	ActCol				: DINT;
	ActVarConfig		: CSV_Config;
	ActVarValueString	: STRING;
	AdressOffset		: DINT;

	FPStart				: R_TRIG;
	FNStart				: F_TRIG;

	FBFileOpen			: FB_FileOpen;
	nOpenMode			: DWORD;
	hHandle				: UINT;

	CreateHeaderLineNow:BOOL;

	FBFileWrite			: FB_FileWrite;
	FBFileClose			: FB_FileClose;
	FileOpenWasBusy		: BOOL;
	FileWriteWasBusy	: BOOL;
	FileCloseWasBusy	: BOOL;
	FileOpenStart		: BOOL;
	FileWriteStart		: BOOL;
	FileCloseStart		: BOOL;

	TempString			: STRING[255];
END_VAR
FPStart(CLK:= nInExport );
FNStart(CLK:= nInExport );

IF 	FPStart.Q THEN
	WorkingStep:=1;
	FileOpenWasBusy:=FALSE;
	FileWriteWasBusy:=FALSE;
	FileCloseWasBusy:=FALSE;
	FileOpenStart:=FALSE;
	FileWriteStart:=FALSE;
	FileCloseStart:=FALSE;
	WorkingStepWriteLine:=1;
	TempString:='';
END_IF;

IF 	FNStart.Q AND WorkingStep<>50 THEN
	WorkingStep:=0;
END_IF


CASE WorkingStep OF

	1:	(* Check File Exist *)
		FindFile_.bExecute:=TRUE;
		IF 	FindFile_.bBusy THEN
			WorkingStep:=2;
		END_IF
	2:
		FindFile_.bExecute:=TRUE;
		IF 	NOT FindFile_.bBusy THEN
			WorkingStep:=3;
		END_IF
	3:
		IF  	filesList_.sFileName='' THEN
			(* Create Header *)
			WorkingStep:=20;
			CreateHeaderLineNow:=CreateHeaderLine;
		ELSIF
			filesList_.sFileName<>'' THEN
			(* File Exists *)
			WorkingStep:=20;
			CreateHeaderLineNow:=FALSE;
		END_IF

	20: (* Open File *)
		IF 	OverwriteExistingFile THEN
			nOpenMode:=FOPEN_MODEWRITE OR FOPEN_MODETEXT ;
		ELSE
			nOpenMode:=FOPEN_MODEAPPEND OR FOPEN_MODETEXT ;
		END_IF
		FBFileOpen(
			sNetId			:= localAMSNetID,
			sPathName	:= strInFileName,
			nMode			:= nOpenMode,
			ePath			:= PATH_GENERIC,
			bExecute		:= FileOpenStart,
			tTimeout		:= t#1s);
			hHandle:=FBFileOpen.hFile;
		FileOpenStart:= TRUE;
		IF 	FBFileOpen.bBusy THEN
			FileOpenWasBusy:=TRUE;
		END_IF
		IF 	NOT FBFileOpen.bBusy AND FileOpenWasBusy THEN
			WorkingStep:=21;
			FileOpenStart:= FALSE;
		END_IF

	21:	(* Write Header if required *)
		IF 	CreateHeaderLineNow THEN
			IF 	WorkingStepWriteLine=0 THEN
				WorkingStepWriteLine:=0;
				TempString:='';
			END_IF

			CASE WorkingStepWriteLine OF
				0: (*Create new CSV config*)
						WorkingStepWriteLine:=1;
				1: (* Open File *)
					FOR ActCol := 1 TO iInNumberOfColumns DO
						(*CSV-Configuration zuweisen*)
						ActVarConfig:=CSVConfig[ActCol];
						TempString:=CONCAT(TempString,ActVarConfig.ColName);
						IF 	ActCol<iInNumberOfColumns THEN
							TempString:=CONCAT(TempString,';');
						ELSE
							TempString:=CONCAT(TempString, '$N');
						END_IF
					END_FOR;
					WorkingStepWriteLine:=2;
				2:(* Write Line *)
				FBFileWrite(
					sNetId				:=localAMSNetID ,
					hFile				:=hHandle ,
					pWriteBuff			:=ADR(TempString) ,
					cbWriteLen			:=LEN(TempString) ,
					bExecute			:=FileWriteStart ,
					tTimeout				:=t#1s );
					FileWriteStart			:= TRUE;
	
				IF 	FBFileWrite.bBusy  THEN
					FileWriteWasBusy:=TRUE;
				END_IF
				IF 	(NOT FBFileWrite.bBusy) AND FileWriteWasBusy THEN
					FileWriteStart:= FALSE;
					FileWriteWasBusy:=FALSE;

					WorkingStepWriteLine:=0;
					WorkingStep:=30;
				END_IF
			END_CASE
		ELSE
			WorkingStep:=30;
		END_IF

	30:	(* Write Data *)
		IF 	WorkingStepWriteLine=0 THEN
			WorkingStepWriteLine:=0;
			TempString:='';
		END_IF

		CASE WorkingStepWriteLine OF
			0: (*Create new CSV config*)
					WorkingStepWriteLine:=1;
			1: (* Open File *)
				FOR ActCol := 1 TO iInNumberOfColumns DO
					(*CSV-Configuration zuweisen*)
					ActVarConfig:=CSVConfig[ActCol];
					AdressOffset:=0;
					ActVarValueString:=TYPEDEF_TO_STRING(ActVarConfig,AdressOffset);
					TempString:=CONCAT(TempString,ActVarValueString);
					IF 	ActCol<iInNumberOfColumns THEN
						TempString:=CONCAT(TempString,';');
					ELSE
						TempString:=CONCAT(TempString, '$N');
					END_IF
				END_FOR
				WorkingStepWriteLine:=2;
			2:(* Write Line *)
			FBFileWrite(
				sNetId				:=localAMSNetID ,
				hFile				:=hHandle ,
				pWriteBuff			:=ADR(TempString) ,
				cbWriteLen			:=LEN(TempString) ,
				bExecute			:=FileWriteStart ,
				tTimeout				:=t#1s );
				FileWriteStart			:= TRUE;

			IF 	FBFileWrite.bBusy  THEN
				FileWriteWasBusy:=TRUE;
			END_IF
			IF 	(NOT FBFileWrite.bBusy) AND FileWriteWasBusy THEN
				FileWriteStart:= FALSE;
				FileWriteWasBusy:=FALSE;

				WorkingStepWriteLine:=0;
				WorkingStep:=40;

			END_IF
		END_CASE

	40: (* Close File *)
		FBFileClose(
			sNetId:=localAMSNetID ,
			hFile:= hHandle,
			bExecute:=FileCloseStart ,
			tTimeout:= t#1s);
		FileCloseStart:=TRUE;
		IF 	FBFileClose.bBusy THEN
			FileCloseWasBusy:=TRUE;
		END_IF

		IF 	NOT FBFileClose.bBusy AND FileCloseWasBusy THEN
			WorkingStep:=50;
		END_IF
	50:(* Done *)
		Done:=TRUE;
		IF 	FNStart.Q THEN
			WorkingStep:=0;
			done:=FALSE;
		END_IF

END_CASE

FindFile_(
	sNetId:= '',
	sPathName:= strInFileName,
	stFindFile=> filesList_
);

FindFile_.bExecute:=FALSE;
END_FUNCTION_BLOCK

(* POU zLibrary/CSV_ImportExport/TYPEDEF_TO_STRING, ST *)
FUNCTION TYPEDEF_TO_STRING : STRING
VAR_INPUT
	TypeData				:CSV_Config;
	inAdressOffset			:DINT;
END_VAR
VAR
	pBOOL					:POINTER TO 	BOOL;
	pBYTE					:POINTER TO 	BYTE;
	pWORD				:POINTER TO 	WORD;
	pDWORD				:POINTER TO 	DWORD;
	pSINT					:POINTER TO 	SINT;
	pUSINT					:POINTER TO USINT;
	pINT					:POINTER TO INT;
	pUINT					:POINTER TO UINT;
	pDINT					:POINTER TO DINT;
	pUDINT				:POINTER TO UDINT;
	pREAL					:POINTER TO REAL;
	pLREAL				:POINTER TO LREAL;
	pSTRING				:POINTER TO STRING(255);
	pTIME					:POINTER TO TIME;
	pTOD					:POINTER TO TOD;
	pDATE					:POINTER TO DATE;
	pDT					:POINTER TO DT;
END_VAR
VAR CONSTANT
	TempTypeData			:DataTypeDef;
END_VAR
IF 	TypeData.ColDataType = TempTypeData.iBOOL THEN
	pBOOL:=TypeData.ColSourceAdr + inAdressOffset;
	TYPEDEF_TO_STRING:=BOOL_TO_STRING(pBOOL^);
ELSIF
	TypeData.ColDataType = TempTypeData.iBYTE THEN
	pBYTE:=TypeData.ColSourceAdr + inAdressOffset;
	TYPEDEF_TO_STRING:=BYTE_TO_STRING(pBYTE^);
ELSIF
	TypeData.ColDataType = TempTypeData.iWORD THEN
	pWORD:=TypeData.ColSourceAdr + inAdressOffset;
	TYPEDEF_TO_STRING:=WORD_TO_STRING(pWORD^);
ELSIF
	TypeData.ColDataType = TempTypeData.iDWORD THEN
	pDWORD:=TypeData.ColSourceAdr + inAdressOffset;
	TYPEDEF_TO_STRING:=DWORD_TO_STRING(pDWORD^);
ELSIF
	TypeData.ColDataType = TempTypeData.iSINT THEN
	pSINT:=TypeData.ColSourceAdr + inAdressOffset;
	TYPEDEF_TO_STRING:=SINT_TO_STRING(pSINT^);
ELSIF
	TypeData.ColDataType = TempTypeData.iUSINT THEN
	pUSINT:=TypeData.ColSourceAdr + inAdressOffset;
	TYPEDEF_TO_STRING:=USINT_TO_STRING(pUSINT^);
ELSIF
	TypeData.ColDataType = TempTypeData.iINT THEN
	pINT:=TypeData.ColSourceAdr + inAdressOffset;
	TYPEDEF_TO_STRING:=INT_TO_STRING(pINT^);
ELSIF
	TypeData.ColDataType = TempTypeData.iUINT THEN
	pUINT:=TypeData.ColSourceAdr + inAdressOffset;
	TYPEDEF_TO_STRING:=UINT_TO_STRING(pUINT^);
ELSIF
	TypeData.ColDataType = TempTypeData.iDINT THEN
	pDINT:=TypeData.ColSourceAdr + inAdressOffset;
	TYPEDEF_TO_STRING:=DINT_TO_STRING(pDINT^);
ELSIF
	TypeData.ColDataType = TempTypeData.iUDINT THEN
	pUDINT:=TypeData.ColSourceAdr + inAdressOffset;
	TYPEDEF_TO_STRING:=UDINT_TO_STRING(pUDINT^);
ELSIF
	TypeData.ColDataType = TempTypeData.iREAL THEN
	pREAL:=TypeData.ColSourceAdr + inAdressOffset;
	TYPEDEF_TO_STRING:=REAL_TO_STRING(pREAL^);
ELSIF
	TypeData.ColDataType = TempTypeData.iLREAL THEN
	pLREAL:=TypeData.ColSourceAdr + inAdressOffset;
	TYPEDEF_TO_STRING:=LREAL_TO_STRING(pLREAL^);
ELSIF
	TypeData.ColDataType = TempTypeData.iSTRING THEN
	pSTRING:=TypeData.ColSourceAdr + inAdressOffset;
	IF 	pSTRING^='' THEN
		TYPEDEF_TO_STRING:='empty';
	ELSE
		TYPEDEF_TO_STRING:=pSTRING^;
	END_IF
ELSIF
	TypeData.ColDataType = TempTypeData.iTIME THEN
	pTIME:=TypeData.ColSourceAdr + inAdressOffset;
	TYPEDEF_TO_STRING:=TIME_TO_STRING(pTIME^);
ELSIF
	TypeData.ColDataType = TempTypeData.iTOD THEN
	pTOD:=TypeData.ColSourceAdr + inAdressOffset;
	TYPEDEF_TO_STRING:=TOD_TO_STRING(pTOD^);
ELSIF
	TypeData.ColDataType = TempTypeData.iDATE THEN
	pDATE:=TypeData.ColSourceAdr + inAdressOffset;
	TYPEDEF_TO_STRING:=DATE_TO_STRING(pDATE^);
ELSIF
	TypeData.ColDataType = TempTypeData.iDT THEN
	pDT:=TypeData.ColSourceAdr + inAdressOffset;
	TYPEDEF_TO_STRING:=DT_TO_SPECIALSTRING(pDT^);
ELSE
	TYPEDEF_TO_STRING:='error';
END_IF
END_FUNCTION

(* POU zLibrary/CSV_ImportExport/DT_TO_SPECIALSTRING, ST *)
FUNCTION DT_TO_SPECIALSTRING : STRING
VAR_INPUT
	inDT			:DT;
END_VAR
VAR
	TempString		:STRING;
	SysTime		:TIMESTRUCT;

	wYear			:WORD;
	wMonth			:WORD;
	wDay			:WORD;
	wHour			:WORD;
	wMin			:WORD;
	wSec			:WORD;
END_VAR
SysTime:=DT_TO_SYSTEMTIME(inDT);
wYear:=SysTime.wYear;
wMonth:=SysTime.wMonth;
wDay:=SysTime.wDay;
wHour:=SysTime.wHour;
wMin:=SysTime.wMinute;
wSec:=SysTime.wSecond;
TempString:='';

IF 	wDay<10 THEN
	TempString:=CONCAT(TempString ,WORD_TO_STRING(0));
END_IF
TempString:=CONCAT(TempString ,WORD_TO_STRING(wDay));
TempString:=CONCAT(TempString , '.');
IF 	wMonth<10 THEN
	TempString:=CONCAT(TempString ,WORD_TO_STRING(0));
END_IF
TempString:=CONCAT(TempString ,WORD_TO_STRING(wMonth));
TempString:=CONCAT(TempString , '.');
TempString:=CONCAT(TempString ,WORD_TO_STRING(wYear));
TempString:=CONCAT(TempString , ' ');
IF 	wHour<10 THEN
	TempString:=CONCAT(TempString ,WORD_TO_STRING(0));
END_IF
TempString:=CONCAT(TempString ,WORD_TO_STRING(wHour));
TempString:=CONCAT(TempString , ':');
IF 	wMin<10 THEN
	TempString:=CONCAT(TempString ,WORD_TO_STRING(0));
END_IF
TempString:=CONCAT(TempString ,WORD_TO_STRING(wMin));
TempString:=CONCAT(TempString , ':');
IF	wSec<10 THEN
	TempString:=CONCAT(TempString ,WORD_TO_STRING(0));
END_IF
TempString:=CONCAT(TempString ,WORD_TO_STRING(wSec));
DT_TO_SPECIALSTRING:=TempString;
END_FUNCTION

(* POU System/Error_and_Message/MessageHandler, ST *)
PROGRAM MessageHandler
VAR_INPUT
	Prio					: DINT; 					(*1=highest, .. , 4=lowest*)
	Btn1Addr 			: POINTER TO BOOL;	(*Address of Button1 , if Zero then Button is unvisible*)
	Btn2Addr 			: POINTER TO BOOL;	(*Address of Button2 , if Zero then Button is unvisible*)
	Msg				: sMessageText;
	MessageLine		: ARRAY [1..10] OF sMessageLine;
	MsgButton1Text		: STRING(20);
	MsgButton2Text		: STRING(20);

	FB_ReadXmlLineMsg	:FB_ReadXmlLine;
END_VAR
VAR_IN_OUT
	sVisu				: sMessageVisu;
END_VAR
VAR_OUTPUT
	MessageActive		: BOOL;
END_VAR
VAR
	EmptyMsg			: sMessageText;
	TempMsg			: sMessageText;
	TempPrio			: DINT;
	MessageGoneFlag	: F_TRIG;
	MessageShowFlag	: R_TRIG;
	Idx, i					: DINT;
	BackupVisu			: STRING;
	ShowVisuMessage	: BOOL;
	VisuMessageActivT	: TON;

	Button1				: VisuButton;
	Button2				: VisuButton;
	btnHide				: VisuButton;
	btnShow			: VisuButton;
	ShowText			: STRING(255);
	LaufschriftShowText	: FB_Laufschrift_STR255;

(* Vars for Disabling Multiselection *)
	Index			: DINT;
	Index_Clear			: DINT;
	FP_MsgLineBool	: ARRAY[1..20] OF R_TRIG;
	LastPressedLine		: DINT;

	Error				: ErrorStruct;
	ErrorPuls			: BOOL:=FALSE;

END_VAR
(*Das ist noch Baustelle!
Es gibt 2 Möglichkeiten:
a) Prio bei Messages mit Button gibt es nicht.
   Wenn eine Meldung mit Button angezeigt wird, dann solange bis diese quittiert ist.
   Dann erst kommt die nächste dran.

b) Jede Meldung mit Button erhält eine eindeutige PLCID.
   Die Visu schreibt für die angezeigte Meldung die ID zurück in VisuID.
   Wenn das Button-Signal in der PLC ankommt werden die IDs verglichen,
   und nur bei VisuID=PLCID wird der Button an die Aufrufstelle weitergereicht.
*)

Lng();

IF 	(NOT TempMsg.ShowMessage OR
	 Msg.Name=TempMsg.Name AND Msg.Text=TempMsg.Text) THEN
	IF 	Msg.Name=TempMsg.Name	AND
		Msg.Text=TempMsg.Text THEN
		IF 	Btn1Addr<>0 THEN
			IF 	MsgButton1Text='' THEN
				MsgButton1Text:='OK';
			END_IF
			Button1.Enable:=TRUE;
			Button1.Visible:=TRUE;
			Button1.TextOn:=MsgButton1Text;
			IF 	sVisu.Button1.Pressed THEN
				Btn1Addr^:=TRUE;
				MessageLine:=sVisu.MessageLine;
				TempMsg.ShowMessage:=FALSE;
			END_IF
		ELSE
			Button1.Visible:=FALSE;
		END_IF

		IF 	Btn2Addr<>0 THEN
			IF 	MsgButton2Text='' THEN
				MsgButton2Text:='Cancel';
			END_IF
			Button2.Enable:=TRUE;
			Button2.Visible:=TRUE;
			Button2.TextOn:=MsgButton2Text;
			IF 	sVisu.Button2.Pressed THEN
				Btn2Addr^:=TRUE;
				TempMsg.ShowMessage:=FALSE;
			END_IF
		ELSE
			Button2.Visible:=FALSE;
		END_IF
	ELSE
		TempMsg:=Msg;
		sVisu.MessageLine:=MessageLine;
	END_IF
	TempMsg.ShowMessage:=TRUE;
	TempPrio:=Prio;

	IF 	NOT ErrorPuls OR
		Error.DateTime = ErrorHandler.EmptyError.DateTime THEN
		Error.DateTime	:= gVarDTSystemtime;
		ErrorPuls 		:= TRUE;
	END_IF
	Error.Text	:= CONCAT('MessageHandler: ',Msg.Text);
	Error.No		:= 1;
	Error.Typ	:= 1;			(* 0=red 1:=orange 2:=blue *)

	IF 	Error.Text<>'' AND
		ST_Lng.b_EndChangeLng THEN
		ErrorHandler.AddError(	ErrorToAdd:=Error,
								sVisu:=Visu.ErrorHandler);
	END_IF
END_IF


(*Clear Input-Var*)
Prio:=0;
Btn1Addr:=0;
Btn2Addr:=0;
Msg:=EmptyMsg;
MsgButton1Text:='';
MsgButton2Text:='';
END_PROGRAM
ACTION ClearAll:
IF NOT sVisu.ShowMessage THEN
	TempPrio:=0;
	TempMsg.Name:='';
	TempMsg.Text:='';
	TempMsg.ID:='';
	TempMsg.ShowMessage:=FALSE;
	TempMsg.Color:=0;
	TempMsg.Station:=0;
	TempMsg.Button1.Visible:=FALSE;
	TempMsg.Button2.Visible:=FALSE;
ELSE
	TempMsg.ShowMessage:=FALSE;
END_IF

(* Copy from visu *)
MessageLine:=sVisu.MessageLine;
END_ACTION
ACTION ClearMessageLines:
FOR idx:=1 TO 10 DO
	MessageHandler.MessageLine[idx].Visible:=FALSE;
	MessageHandler.MessageLine[idx].Editable:=FALSE;
	MessageHandler.MessageLine[idx].Text:='';
	MessageHandler.MessageLine[idx].MsgInt:=0;
	MessageHandler.MessageLine[idx].MsgBool:=FALSE;
	MessageHandler.MessageLine[idx].MsgReal:=0.0;
	MessageHandler.MessageLine[idx].MsgString:='';
	MessageHandler.MessageLine[idx].MsgTypeEnum:=MsgDataTypeNone;
END_FOR
END_ACTION
ACTION DisableMultiSelect:
LastPressedLine:=0;

FOR Index:=1 TO 10 DO
	FP_MsgLineBool[Index](CLK:=sVisu.MessageLine[Index].MsgBool);
	IF FP_MsgLineBool[Index].Q THEN
		LastPressedLine:=Index;
		EXIT;
	END_IF
END_FOR

IF LastPressedLine>0 THEN

	FOR Index_Clear:=1 TO 10 DO
		MessageLine[Index_Clear].MsgBool:=(LastPressedLine=Index_Clear);
	END_FOR

END_IF
END_ACTION
ACTION Lng:
IF	TempMsg.ID <> '' THEN

	FB_ReadXmlLineMsg(
		Prefix:= 'MSG',
		ID:= TempMsg.ID,
		File:= 'MSG.xml',
		Text=>);

	IF 	FB_ReadXmlLineMsg.Text <> ''  THEN
		TempMsg.Text:=CONCAT(TempMsg.ID,':$N$R');
		TempMsg.Text:=CONCAT(TempMsg.Text,FB_ReadXmlLineMsg.Text);
		Msg.Text:=TempMsg.Text;

		ShowText:=CONCAT(TempMsg.ID,': ');
		ShowText:=CONCAT(ShowText,FB_ReadXmlLineMsg.Text);
		FOR i:=1 TO 10 DO
			IF	FIND(ShowText, '$N') > 0 THEN
				ShowText:=DELETE (ShowText,1,FIND(ShowText, '$N'));
			END_IF
			IF	FIND(ShowText, '$R') > 0 THEN
				ShowText:=DELETE (ShowText,1,FIND(ShowText, '$R'));
			END_IF
		END_FOR
		IF LEN(ShowText) > 60 THEN
			ShowText:=CONCAT(ShowText,' ->   ');
		END_IF
		LaufschriftShowText(
				N:= 60,
				StepWidth:=1,
				PT:= t#100ms ,
				Text:= ShowText,
				Display=>BtnShow.TextOn
				);
	ELSE
		TempMsg.Text:=CONCAT(TempMsg.ID,':..... ');
	END_IF
ELSE
	ShowText:=TempMsg.Text;
	FOR i:=1 TO 10 DO
		IF	FIND(ShowText, '$N') > 0 THEN
			ShowText:=DELETE (ShowText,1,FIND(ShowText, '$N'));
		END_IF
		IF	FIND(ShowText, '$R') > 0 THEN
			ShowText:=DELETE (ShowText,1,FIND(ShowText, '$R'));
		END_IF
	END_FOR
	IF LEN(ShowText) > 60 THEN
		ShowText:=CONCAT(ShowText,' ->   ');
	END_IF
	LaufschriftShowText(
			N:= 60,
			StepWidth:=1,
			PT:= t#100ms ,
			Text:= ShowText,
			Display=>BtnShow.TextOn
			);
END_IF
END_ACTION
ACTION VisuUpdate:
sVisu.Name:=TempMsg.Name;
sVisu.Text:=TempMsg.Text;
sVisu.ID:=TempMsg.ID;
sVisu.ShowMessage:=TempMsg.ShowMessage;
sVisu.Color:=TempMsg.Color;
sVisu.Station:=TempMsg.Station;

sVisu.Button1:=TempMsg.Button1;
sVisu.Button2:=TempMsg.Button2;


(* Write to visu *)

sVisu.MessageLine:=MessageLine;
FOR idx:=1 TO 10 DO
	CASE sVisu.MessageLine[idx].MsgTypeEnum OF
		MsgDataTypeBool: sVisu.MessageLine[idx].MsgType:='BOOL';
		MsgDataTypeDint: sVisu.MessageLine[idx].MsgType:='DINT';
		MsgDataTypeReal: sVisu.MessageLine[idx].MsgType:='REAL';
		MsgDataTypeString: sVisu.MessageLine[idx].MsgType:='STRING';
	ELSE
		sVisu.MessageLine[idx].MsgType:='';
	END_CASE
END_FOR

MessageGoneFlag(CLK:=sVisu.ShowMessage);
MessageShowFlag(CLK:=sVisu.ShowMessage AND NOT sVisu.BtnShow.Pressed);

(*Meldefenster öffnen, wenn Meldung neu aktiv wird (als Impuls)*)
IF MessageShowFlag.Q AND CurrentVisu<>'ZLIB_VISUMESSAGEHANDLER' THEN
	ShowVisuMessage:=TRUE;
	BackupVisu:=CurrentVisu;
END_IF
VisuMessageActivT(IN:=CurrentVisu='ZLIB_VISUMESSAGEHANDLER' ,PT:=T#1s);
IF 	CurrentVisu='ZLIB_VISUMESSAGEHANDLER'AND
	ShowVisuMessage THEN
	ShowVisuMessage:=FALSE;
END_IF
IF 	ShowVisuMessage THEN
	CurrentVisu:='ZLIB_VISUMESSAGEHANDLER';
END_IF

(*Button "Meldung einblenden" anzeigen, wenn Meldung aktiv aber Meldefenster nicht offen*)
IF 	sVisu.ShowMessage AND
	CurrentVisu<>'ZLIB_VISUMESSAGEHANDLER' AND
	NOT ShowVisuMessage THEN
	BtnShow.Visible:=TRUE;
	BtnShow.Enable:=TRUE;
	BtnShow.ButtBackColor:=Visu.Message.Color;
ELSE
	BtnShow.Visible:=FALSE;
END_IF

(*Button "Minimieren" einblenden, wenn Meldefenster offen*)
IF 	CurrentVisu='ZLIB_VISUMESSAGEHANDLER' THEN
	BtnHide.Visible:=TRUE;
	BtnHide.Enable:=TRUE;
	BtnHide.TextOn:='Meldung minimieren';
	BtnHide.ButtBackColor:=Color.control;
ELSE
	BtnHide.Visible:=FALSE;
END_IF

(*Meldefenster komplett schliessen, wenn keine Meldung mehr ansteht*)
IF 	MessageGoneFlag.Q OR
	BtnHide.Pressed THEN
	IF 	BackupVisu<>'' OR
		BackupVisu='ZLIBVISUMESSAGEHANDLER'THEN
		CurrentVisu:=BackupVisu;
	ELSE
		CurrentVisu:='MAIN';
	END_IF
END_IF;

MessageActive := sVisu.ShowMessage OR sVisu.BtnShow.Visible;


(*VisuButton Handler Call*)
Button1(	Button:= TempMsg.Button1);
Button2(	Button:= TempMsg.Button2);
btnHide(	Button:= sVisu.btnHide);
btnShow(	Button:= sVisu.btnShow);
END_ACTION

(* POU zLibrary/ept/Sprache/FB_ReadXmlLine, ST *)
FUNCTION_BLOCK FB_ReadXmlLine
VAR_INPUT
	Prefix					: STRING;
	ID						: STRING;
	File						: STRING;
END_VAR
VAR_OUTPUT
	Text					: STRING(255);
END_VAR

VAR
	bError							: BOOL;
	nErrId							: UDINT;

	fb_state_entry					: ST_StateEntry;

	CURRENTLANGUAGECopy			: STRING(5);
	IdCopy							: STRING;
END_VAR
(*======================================================
   ST: FB_ReadXmlLine
 ------------------------------------------------------
   Auth: 	Werner Frield    						 
   Date: 	23.12.2020    						     
   Rev.: 		1.0	
   Desc	
	-	Mit diesem FB kann Srachabängig ein Text aus einer xml Datei ausgelesen werden		
	-	Das Programm ST_ReadXmlLine wird zum auslesen benutzt.
	-	Die XML Datei muss im PLC Verzeichnis unter TRANS abgelegt werden und 
		mit der Excel Datei (_Texte.xlsm) erstellt werden.
	-	abhängig von der CURRENTLANGUAGE werden Srachabängig die Texte ausgelesen

Beispiel:
FB_ReadXmlLineConf(
	Prefix:= 'CONFIG',			(*erste Spalte der Excel Datei*)
	ID:= 'ST03_473_B70_0',		(*zweite Spalte der Excel Datei*)
	File:= 'CONFIG.xml',		(* xml Datei Name*)
	Text=> );					(* hier kommt der passende Text zurück. abhängig von der angewählten Sprache (DE, EN,CZ*)

 ========================================================*)
fb_state_entry(i16_pos:= 1);
CASE fb_state_entry.i16_step OF
(*=======================================================*)
INIT_OBJ:

	(*-----------------------Weiterschaltbedingungen----------------------------*)
	fb_state_entry.i16_next_step:=INIT;

(*=======================================================*)
INIT:
	IF	TD.ArtNo <> '' AND CURRENTLANGUAGE <> '' THEN
		fb_state_entry.i16_next_step:=BEREIT;
	END_IF

(*=======================================================*)
BEREIT:	fb_state_entry.s_debugtext:='warte auf Start';

	IF	fb_state_entry.E THEN
		bError:=FALSE;
		IdCopy:= ID;
	END_IF
	IF	Prefix <> '' AND ID <> '' AND
		ST_ReadXmlLine.b_ready THEN

		IF	CURRENTLANGUAGECopy <> CURRENTLANGUAGE OR
			IdCopy <> ID THEN
			IF	Prefix <> 'MSG' THEN
				fb_state_entry.i16_next_step:=110;		(*ST_ReadXmlLine*)
			ELSE
				fb_state_entry.i16_next_step:=210;		(*ST_ReadXmlLineMsg*)
			END_IF
		END_IF
	END_IF

	IF	fb_state_entry.X THEN
		CURRENTLANGUAGECopy := CURRENTLANGUAGE;
		Text:='';
	END_IF

(*=======================================================*)
110:  fb_state_entry.s_debugtext:='*Warten bis Lesen erlaubt ist';

	IF	TestAndSet(ST_ReadXmlLine.LockFlag) THEN
		fb_state_entry.i16_next_step := 120;
	END_IF

	IF	fb_state_entry.X THEN
		ST_ReadXmlLine.b_start:=TRUE;
		ST_ReadXmlLine.s_Prefix:= Prefix;
		ST_ReadXmlLine.s_ID:= ID;
		ST_ReadXmlLine.s_File:= File;
		ST_ReadXmlLine.s_Text;
	END_IF

(*=======================================================*)
120:  fb_state_entry.s_debugtext:='*Warten auf busy';

	IF 	ST_ReadXmlLine.b_busy THEN
		fb_state_entry.i16_next_step := 130;
	ELSIF
		fb_state_entry.fb_ton_Step.ET > t#3000ms THEN
		nErrId := ST_ReadXmlLine.nErrId;
		fb_state_entry.s_debugtext:='timeout';
		fb_state_entry.i16_next_step := FEHLER;
	END_IF

(*=======================================================*)
130:  fb_state_entry.s_debugtext:='*Warten auf fertig';

	IF 	ST_ReadXmlLine.b_done THEN
		text:=ST_ReadXmlLine.s_Text;

		fb_state_entry.i16_next_step := BEREIT;
	ELSIF
		fb_state_entry.fb_ton_Step.ET > t#3000ms THEN
		nErrId := ST_ReadXmlLine.nErrId;
		fb_state_entry.s_debugtext:='timeout';
		fb_state_entry.i16_next_step := FEHLER;
	END_IF

(*=======================================================*)
(*=======================================================*)
210:  fb_state_entry.s_debugtext:='*Warten bis Lesen erlaubt ist';

	IF	TestAndSet(ST_ReadXmlLineMsg.LockFlag) THEN
		fb_state_entry.i16_next_step := 220;
	END_IF

	IF	fb_state_entry.X THEN
		ST_ReadXmlLineMsg.b_start:=TRUE;
		ST_ReadXmlLineMsg.s_Prefix:= Prefix;
		ST_ReadXmlLineMsg.s_ID:= ID;
		ST_ReadXmlLineMsg.s_File:= File;
		ST_ReadXmlLineMsg.s_Text;
	END_IF

(*=======================================================*)
220:  fb_state_entry.s_debugtext:='*Warten auf busy';

	IF 	ST_ReadXmlLineMsg.b_busy THEN
		fb_state_entry.i16_next_step := 230;
	ELSIF
		fb_state_entry.fb_ton_Step.ET > t#3000ms THEN
		nErrId := ST_ReadXmlLineMsg.nErrId;
		fb_state_entry.s_debugtext:='timeout';
		fb_state_entry.i16_next_step := FEHLER;
	END_IF

(*=======================================================*)
230:  fb_state_entry.s_debugtext:='*Warten auf fertig';

	IF 	ST_ReadXmlLineMsg.b_done THEN
		text:=ST_ReadXmlLineMsg.s_Text;
		fb_state_entry.i16_next_step := BEREIT;
	ELSIF
		fb_state_entry.fb_ton_Step.ET > t#3000ms THEN
		nErrId := ST_ReadXmlLineMsg.nErrId;
		fb_state_entry.s_debugtext:='timeout';
		fb_state_entry.i16_next_step := FEHLER;
	END_IF

(*=======================================================*)
FEHLER:
	IF 	fb_state_entry.E THEN
		bError:=TRUE;
		Text:=ST_ReadXmlLine.s_Text;
	END_IF

	fb_state_entry.s_debugtext:='nErrorID: ';
	fb_state_entry.s_debugtext:=CONCAT(fb_state_entry.s_debugtext, UDINT_TO_STRING(nErrId));
	fb_state_entry.i16_next_step:=BEREIT;

END_CASE
fb_state_entry(i16_pos:= 2);
END_FUNCTION_BLOCK

(* POU zLibrary/ept/Funktionsbausteine/ST_StateEntry, ST *)
FUNCTION_BLOCK ST_StateEntry
VAR
	arr_last_step_history	: ARRAY[0..31] OF STRING(110);
	last_pos 			: INT := 0;
	interner_step		: INT := 0;
	s_stepTime 			: STRING;
END_VAR
VAR_OUTPUT
	i16_last_step 			: enum_step_nr := INIT_OBJ;	(* Der Schritt vor diesem Schritt *)
	i16_step 				: enum_step_nr := INIT_OBJ;	(* Diese variable soll vom "case step of" verwendet werden *)
	E					: BOOL;					(* Aktiv bei betreten des Steps *)
	X					: BOOL;					(* Aktiv beim verlassen des Steps *)
	b_error 				: BOOL := FALSE;			(* Ablauf Pos 1,2,1,2,1,2,... nicht richtig *)
	fb_ton_Step			: TON;
END_VAR
VAR_INPUT
	i16_next_step 		: enum_step_nr := INIT_OBJ;	(* Nächster schritt *)
	i16_pos 				: INT;					(* Pos = 1: Aufruf vor dem Case step of ---  Pos = 2: Aufruf nach dem Case step of*)
	s_debugtext			: STRING(100);
END_VAR
VAR_TEMP
	i					: INT := 0;
END_VAR
VAR CONSTANT
	t_MaxStepTime		: TIME := T#60S;
END_VAR
(*stepTime ermitteln*)
fb_ton_Step(IN:= , PT:=fb_ton_Step.ET + t#10s , Q=>  , ET=> );
IF	i16_step = i16_next_step THEN
	fb_ton_Step.IN:=TRUE;
END_IF

IF	NOT b_error THEN
	CASE interner_step OF
		0:
			(* Mitten im Schritt drin *)
			X := FALSE;
			E := FALSE;


			(* Schritt wird verlassen *)
			IF i16_step <> i16_next_step AND i16_pos = 1 THEN
				subrDebugtext();
				interner_step := 10;
				X := TRUE;
				E := FALSE;
				fb_ton_Step.IN:=FALSE;
			END_IF

		10:
			(* Eintritt in neuen Schritt *)
			IF i16_pos = 1 THEN
				X := FALSE;
				E := TRUE;

				(* Schalte Schritt weiter *)
				i16_last_step := i16_step;
				i16_step := i16_next_step;
				(* Baue Statehistory *)

				IF  E THEN
					FOR i:= 31 TO 1 BY -1 DO
						arr_last_step_history[i] := arr_last_step_history[i-1];
					END_FOR
					arr_last_step_history[0] := '';
					s_stepTime:='';
					s_debugtext:='';
				END_IF

				interner_step := 0;

			END_IF
	END_CASE
END_IF

IF 	(fb_ton_Step.ET >= T#200ms AND arr_last_step_history[0] = '') OR	(* Am Anfang Debugtext schreiben, damit etwas drin steht *)
	(fb_ton_Step.Q AND s_stepTime <> '>1m') THEN	(* Debugtext schreiben, wenn t_MaxStepTime erreicht wird *)
	subrDebugtext();
END_IF

(* Prüfe Baustein *)
IF 	i16_pos = last_pos THEN
	b_error := TRUE;
END_IF

last_pos := i16_pos;
END_FUNCTION_BLOCK
ACTION subrDebugtext:
s_stepTime:=ET_TO_STRING(fb_ton_Step.ET);
IF 	fb_ton_Step.ET >= t_MaxStepTime THEN
	s_stepTime:=CONCAT('>',s_StepTime);
END_IF

(* history zusammenbauen aus StepNr, StepTime und debugtext*)
CASE i16_step OF
	INIT_OBJ :			arr_last_step_history[0]:='INIT_OBJ';
	INIT :				arr_last_step_history[0]:='INIT';
	BEREIT :			arr_last_step_history[0]:='BEREIT';
	HALT :				arr_last_step_history[0]:='HALT';
	STOP :				arr_last_step_history[0]:='STOP';
	FEHLER :			arr_last_step_history[0]:='FEHLER';
	INAKTIV:			arr_last_step_history[0]:='INAKTIV ';
ELSE
	arr_last_step_history[0] := INT_TO_STRING(i16_step);
END_CASE

IF 	s_stepTime ='0ms' OR s_stepTime =''THEN
	s_stepTime:='3ms';		(*damit nicht 0 drin steht*)
END_IF
arr_last_step_history[0] := CONCAT(arr_last_step_history[0],':  ');
arr_last_step_history[0] := CONCAT(arr_last_step_history[0],s_stepTime);
arr_last_step_history[0] := CONCAT(arr_last_step_history[0],': ');
arr_last_step_history[0] := CONCAT(arr_last_step_history[0],s_debugtext);
END_ACTION

(* POU zLibrary/ept/Funktionen/ET_TO_STRING, ST *)
FUNCTION ET_TO_STRING :STRING
VAR_INPUT
	et		:TIME;
END_VAR

VAR

END_VAR
ET_TO_STRING:=TIME_TO_STRING(et);
ET_TO_STRING:=DELETE(ET_TO_STRING,2,1);
END_FUNCTION

(* POU zLibrary/ept/Sprache/ST_ReadXmlLine, ST *)
PROGRAM ST_ReadXmlLine (*Programm wird nur vom FB_ReadXmlLine benutzt*)
VAR_INPUT
	b_start					: BOOL;
	s_Prefix					: STRING;
	s_ID					: STRING;
	s_File					: STRING;
	s_XmlHelp				: T_MaxString;	(* in diese Variable schreibt der XML-Bautstein die ausgelesenen Daten *)
END_VAR
VAR_OUTPUT
	b_EndChangeLng		: BOOL;
	b_busy					: BOOL;
	b_ready					: BOOL;
	b_done					: BOOL;

	s_Text					: STRING(255);
END_VAR

VAR

	LockFlag						: BOOL := FALSE;	(* Ganz wichtig, wenn diese Variable TRUE ist, dann kann die Struktur "Visu.MeldungProduktion" nicht verändert werden *)
	b_Error							: BOOL;
	nErrId							: UDINT;
	s_filePath						: T_MaxString;
	s_Xpath							: T_MaxString;

	fb_state_entry					: ST_StateEntry;
	fb_xml_srv_read					: FB_XmlSrvReadByName;	(* XML Baustein zum Auslesen der CONFIG *)

	CURRENTLANGUAGECopy			: STRING(5);
END_VAR
VAR CONSTANT
	s_SymName					: STRING:='ST_ReadXmlLine.s_XmlHelp';
END_VAR
(*Programm wird nur vom FB_ReadXmlLine benutzt*)

(*===================================================================================================*)
fb_state_entry(i16_pos:= 1);

CASE fb_state_entry.i16_step OF
(*=======================================================*)
INIT_OBJ:

	fb_state_entry.i16_next_step:=INIT;

(*=======================================================*)
INIT:

	IF	TD.ArtNo <> '' THEN
		fb_state_entry.i16_next_step:=BEREIT;
	END_IF

(*=======================================================*)
BEREIT:	fb_state_entry.s_debugtext:='warte auf Start';

	IF	fb_state_entry.E THEN
		b_Error:=FALSE;
		b_ready:=TRUE;
		LockFree();
	END_IF

	IF	s_Prefix <> '' AND s_ID <> '' AND
		b_start THEN
		fb_state_entry.i16_next_step:=110;
(*		LockGet();	(* Ablauf ist immer derselbe, zuerst LockGet, dann Strukturen ändern, dann LockFree *)*)
	END_IF

	IF	fb_state_entry.fb_ton_Step.ET >t#10ms THEN
		b_EndChangeLng:=TRUE;
	END_IF

	IF	fb_state_entry.X THEN
		IF 	CURRENTLANGUAGECopy<>CURRENTLANGUAGE THEN
			CURRENTLANGUAGECopy:=CURRENTLANGUAGE;
			b_EndChangeLng:=FALSE;
		END_IF
		s_XmlHelp:='';
		s_Text:='';
		b_ready:=FALSE;
		b_done:=FALSE;
		b_busy:=TRUE;
	END_IF

(*=======================================================*)
110:	fb_state_entry.s_debugtext:='Zeile aus der XMl auslesen';

	IF	fb_state_entry.E THEN
		s_filePath := CONCAT(s_PLC_path,'TRANS\');
		s_filePath := CONCAT(s_filePath,s_File);

		s_Xpath:= '/dynamic-text/text-list/text[@prefix=$'';
		s_Xpath:=CONCAT(s_Xpath,s_Prefix);
		s_Xpath:=CONCAT(s_Xpath,'$' and @id=$'');
		s_Xpath:=CONCAT(s_Xpath,s_ID);
		s_Xpath:=CONCAT(s_Xpath,'$']/');
		s_Xpath:=CONCAT(s_Xpath, CURRENTLANGUAGE);
	END_IF

	(*-----------------------Weiterschaltbedingungen----------------------------*)
	fb_state_entry.i16_next_step := 120;

(*=======================================================*)
120:	fb_state_entry.s_debugtext:='Starte Daten lesen ';

	IF 	fb_state_entry.E THEN
		fb_xml_srv_read.sFilePath := s_filePath;
		fb_xml_srv_read.sXPath :=s_Xpath;
		fb_xml_srv_read.sSymName := s_SymName;
		fb_xml_srv_read.bExecute := TRUE;
	END_IF

	(*-----------------------Weiterschaltbedingungen----------------------------*)
	IF 	fb_xml_srv_read.bBusy THEN
		fb_xml_srv_read.bExecute := FALSE;
		fb_state_entry.i16_next_step := 130;
	END_IF

(*=======================================================*)
130:fb_state_entry.s_debugtext:='warte auf fertig';

	(*-----------------------Weiterschaltbedingungen----------------------------*)
	IF  	NOT fb_xml_srv_read.bBusy  THEN
		fb_state_entry.i16_next_step := 140;
	ELSIF
		fb_state_entry.fb_ton_Step.ET > t#3000ms THEN
		nErrId := fb_xml_srv_read.nErrId;
		fb_state_entry.s_debugtext:='timeout';
		fb_state_entry.i16_next_step := FEHLER;
	END_IF

(*=======================================================*)
140:fb_state_entry.s_debugtext:='prüfe auf Fehler';

	(*-----------------------Weiterschaltbedingungen----------------------------*)
	IF  	fb_xml_srv_read.bError OR
		s_XmlHelp = '' THEN
		nErrId := fb_xml_srv_read.nErrId;
		fb_state_entry.i16_next_step := FEHLER;
	ELSE
		s_Text:=s_XmlHelp;
		fb_state_entry.i16_next_step := BEREIT;
		b_done:=TRUE;
		b_busy:=FALSE;
	END_IF


(*=======================================================*)
FEHLER:
	IF 	fb_state_entry.E THEN
		b_Error:=TRUE;
		s_Text:='!!! ';
		s_Text:= CONCAT(s_Text,s_Prefix);
		s_Text:= CONCAT(s_Text,'-');
		s_Text:= CONCAT(s_Text,s_ID);
		s_Text:= CONCAT(s_Text,' not found !!!');
	END_IF

	fb_state_entry.s_debugtext:='nErrorID: ';
	fb_state_entry.s_debugtext:=CONCAT(fb_state_entry.s_debugtext, UDINT_TO_STRING(nErrId));
	fb_state_entry.s_debugtext:=CONCAT(fb_state_entry.s_debugtext, ' =>');
	fb_state_entry.s_debugtext:=CONCAT(fb_state_entry.s_debugtext, s_Text);

	(*-----------------------Weiterschaltbedingungen----------------------------*)
	fb_state_entry.i16_next_step:=BEREIT;

	IF 	fb_state_entry.E THEN
		b_done:=TRUE;
		b_busy:=FALSE;
	END_IF

END_CASE

fb_state_entry(i16_pos:= 2);

b_start:=FALSE;


(* XML *)
fb_xml_srv_read(
	sNetId:= '',
	ePath:= PATH_GENERIC,
	nMode:= XMLSRV_SKIPMISSING,
	sSymName:= ,
	sFilePath:= ,
	sXPath:= ,
	bExecute:= ,
	tTimeout:= t#10s,
	bBusy=> ,
	bError=> ,
	nErrId=> );
END_PROGRAM
ACTION LockFree:
LockFlag := FALSE;	(* wieder freigeben *)
END_ACTION
ACTION LockGet:
WHILE NOT TestAndSet(LockFlag) DO	(* Mit der Funktion TestAndSet kann ein Flag nicht unterbrechbar geprüft und gesetzt werden *)
	;	(* Wait until Lock is free *)
END_WHILE
(*LockFlag: Ist ein boolsches Flag, das geprüft wird
 - war es FALSE, dann war das Flag frei und wird gesetzt (blockiert von nun an), die Funktion liefert TRUE
 - war es TRUE, dann war das Flag bereits belegt (blockiert), die Funktion liefert FALSE*)
END_ACTION

(* POU zLibrary/ept/Sprache/ST_ReadXmlLineMsg, ST *)
PROGRAM ST_ReadXmlLineMsg
VAR_INPUT
	b_start					: BOOL;
	s_Prefix					: STRING;
	s_ID					: STRING;
	s_File					: STRING;
	s_XmlHelp				: T_MaxString;	(* in diese Variable schreibt der XML-Bautstein die ausgelesenen Daten *)
END_VAR
VAR_OUTPUT
	b_EndChangeLng		: BOOL;
	b_busy					: BOOL;
	b_ready					: BOOL;
	b_done					: BOOL;

	s_Text					: STRING(255);
END_VAR

VAR
	LockFlag						: BOOL := FALSE;	(* Ganz wichtig, wenn diese Variable TRUE ist, dann kann die Struktur "Visu.MeldungProduktion" nicht verändert werden *)
	b_Error							: BOOL;
	nErrId							: UDINT;
	s_filePath						: T_MaxString;
	s_Xpath							: T_MaxString;

	fb_state_entry					: ST_StateEntry;
	fb_xml_srv_read					: FB_XmlSrvReadByName;	(* XML Baustein zum Auslesen der CONFIG *)

	CURRENTLANGUAGECopy			: STRING(5);
END_VAR
VAR CONSTANT
	s_SymName					: STRING:='ST_ReadXmlLineMsg.s_XmlHelp';
END_VAR
(*===================================================================================================*)
fb_state_entry(i16_pos:= 1);

CASE fb_state_entry.i16_step OF
(*=======================================================*)
INIT_OBJ:

	fb_state_entry.i16_next_step:=INIT;

(*=======================================================*)
INIT:

	IF	TD.ArtNo <> '' THEN
		fb_state_entry.i16_next_step:=BEREIT;
	END_IF

(*=======================================================*)
BEREIT:	fb_state_entry.s_debugtext:='warte auf Start';

	IF	fb_state_entry.E THEN
		b_Error:=FALSE;
		b_ready:=TRUE;
		LockFree();
	END_IF

	IF	s_Prefix <> '' AND s_ID <> '' AND
		b_start THEN
		fb_state_entry.i16_next_step:=110;
(*		LockGet();	(* Ablauf ist immer derselbe, zuerst LockGet, dann Strukturen ändern, dann LockFree *)*)
	END_IF

	IF	fb_state_entry.fb_ton_Step.ET >t#10ms THEN
		b_EndChangeLng:=TRUE;
	END_IF

	IF	fb_state_entry.X THEN
		IF 	CURRENTLANGUAGECopy<>CURRENTLANGUAGE THEN
			CURRENTLANGUAGECopy:=CURRENTLANGUAGE;
			b_EndChangeLng:=FALSE;
		END_IF
		s_XmlHelp:='';
		s_Text:='';
		b_ready:=FALSE;
		b_done:=FALSE;
		b_busy:=TRUE;
	END_IF

(*=======================================================*)
110:	fb_state_entry.s_debugtext:='Zeile aus der XML auslesen';

	IF	fb_state_entry.E THEN
		s_filePath := CONCAT(s_PLC_path,'TRANS\');
		s_filePath := CONCAT(s_filePath,s_File);

		s_Xpath:= '/dynamic-text/text-list/text[@prefix=$'';
		s_Xpath:=CONCAT(s_Xpath,s_Prefix);
		s_Xpath:=CONCAT(s_Xpath,'$' and @id=$'');
		s_Xpath:=CONCAT(s_Xpath,s_ID);
		s_Xpath:=CONCAT(s_Xpath,'$']/');
		s_Xpath:=CONCAT(s_Xpath, CURRENTLANGUAGE);
	END_IF

	(*-----------------------Weiterschaltbedingungen----------------------------*)
	fb_state_entry.i16_next_step := 120;

(*=======================================================*)
120:	fb_state_entry.s_debugtext:='Starte Daten lesen ';

	IF fb_state_entry.E THEN
		fb_xml_srv_read.sFilePath := s_filePath;
		fb_xml_srv_read.sXPath :=s_Xpath;
		fb_xml_srv_read.sSymName := s_SymName;
		fb_xml_srv_read.bExecute := TRUE;
	END_IF

	(*-----------------------Weiterschaltbedingungen----------------------------*)
	IF 	fb_xml_srv_read.bBusy THEN
		fb_xml_srv_read.bExecute := FALSE;
		fb_state_entry.i16_next_step := 130;
	END_IF

(*=======================================================*)
130:fb_state_entry.s_debugtext:='warte auf fertig';

	(*-----------------------Weiterschaltbedingungen----------------------------*)
	IF  	NOT fb_xml_srv_read.bBusy  THEN
		fb_state_entry.i16_next_step := 140;
	ELSIF
		fb_state_entry.fb_ton_Step.ET > t#3000ms THEN
		nErrId := fb_xml_srv_read.nErrId;
		fb_state_entry.s_debugtext:='timeout';
		fb_state_entry.i16_next_step := FEHLER;
	END_IF

(*=======================================================*)
140:fb_state_entry.s_debugtext:='prüfe auf Fehler';

	(*-----------------------Weiterschaltbedingungen----------------------------*)
	IF  	fb_xml_srv_read.bError OR
		s_XmlHelp = '' THEN
		nErrId := fb_xml_srv_read.nErrId;
		fb_state_entry.i16_next_step := FEHLER;
	ELSE
		s_Text:=s_XmlHelp;
		fb_state_entry.i16_next_step := BEREIT;
		b_done:=TRUE;
		b_busy:=FALSE;
	END_IF


(*=======================================================*)
FEHLER:
	IF 	fb_state_entry.E THEN
		b_Error:=TRUE;
		s_Text:='!!! ';
		s_Text:= CONCAT(s_Text,s_Prefix);
		s_Text:= CONCAT(s_Text,'-');
		s_Text:= CONCAT(s_Text,s_ID);
		s_Text:= CONCAT(s_Text,' not found !!!');
	END_IF

	fb_state_entry.s_debugtext:='nErrorID: ';
	fb_state_entry.s_debugtext:=CONCAT(fb_state_entry.s_debugtext, UDINT_TO_STRING(nErrId));
	fb_state_entry.s_debugtext:=CONCAT(fb_state_entry.s_debugtext, ' =>');
	fb_state_entry.s_debugtext:=CONCAT(fb_state_entry.s_debugtext, s_Text);

	(*-----------------------Weiterschaltbedingungen----------------------------*)
	fb_state_entry.i16_next_step:=BEREIT;

	IF 	fb_state_entry.E THEN
		b_done:=TRUE;
		b_busy:=FALSE;
	END_IF

END_CASE

fb_state_entry(i16_pos:= 2);

b_start:=FALSE;


(* XML *)
fb_xml_srv_read(
	sNetId:= '',
	ePath:= PATH_GENERIC,
	nMode:= XMLSRV_SKIPMISSING,
	sSymName:= ,
	sFilePath:= ,
	sXPath:= ,
	bExecute:= ,
	tTimeout:= t#10s,
	bBusy=> ,
	bError=> ,
	nErrId=> );
END_PROGRAM
ACTION LockFree:
LockFlag := FALSE;	(* wieder freigeben *)
END_ACTION
ACTION LockGet:
WHILE NOT TestAndSet(LockFlag) DO	(* Mit der Funktion TestAndSet kann ein Flag nicht unterbrechbar geprüft und gesetzt werden *)
	;	(* Wait until Lock is free *)
END_WHILE
(*LockFlag: Ist ein boolsches Flag, das geprüft wird
 - war es FALSE, dann war das Flag frei und wird gesetzt (blockiert von nun an), die Funktion liefert TRUE
 - war es TRUE, dann war das Flag bereits belegt (blockiert), die Funktion liefert FALSE*)
END_ACTION

(* POU System/VisuInterface/VisuButton, ST *)
FUNCTION_BLOCK VisuButton
VAR_INPUT
	Enable						:	BOOL := TRUE;
	Visible						:	BOOL := TRUE;
	PressedExt				:	BOOL;
	StateOn						:	BOOL;

	TextColEnabled		:	DINT;
	TextColDisabled		:	DINT;
	ButtColOn					:	DINT;
	ButtBackColor 		:	DINT;
	ButtColDisabled		:	DINT;

	TextOn						:	STRING;
	TextOff						:	STRING(30);

END_VAR
VAR_IN_OUT
	Button				: 	sButtonVisu;

END_VAR

VAR_OUTPUT
	PressedFlag	:	BOOL;
	Pressed			:	BOOL;
END_VAR

VAR
	PressedRTrig	:	R_TRIG;


END_VAR

(* Call of FB
	VisuButton(	Button:=Visu.ButtonAuto,
						Enable:=xxxx  ,
						Visible:=TRUE ,
						PressedExt:=FALSE ,
						StateOn:= xxxx,

						TextColEnabled:= 	Color.black ,
						TextColDisabled:=	Color.white ,
						ButtColOff:= 			Color.grey,
						ButtColOn:= 			Color.lime,
						ButtColPressed:=	Color.yellow ,
						ButtColDisabled:=	Color.lightgrey ,

						TextOn:= 'xxxx',
						TextOff:= 'xxxx',
						);
*)
(* Init colors if not filled *)
 IF 	TextColEnabled = 0 THEN
	TextColEnabled:= 	Color.black ;
END_IF
 IF 	TextColDisabled = 0 THEN
	TextColDisabled:= 	Color.darkgrey ;
END_IF

IF 	ButtBackColor = 0 THEN
	ButtBackColor:= 	Color.control ;
END_IF

IF 	ButtColOn = 0 THEN
	ButtColOn:= 	Color.lime ;
END_IF

IF 	ButtColDisabled = 0 THEN
	ButtColDisabled:= 	Color.control ;
END_IF

(* Check Button pressed *)
Pressed:=Button.Pressed OR PressedExt;

(* Flag button pressed *)
PressedRTrig(CLK:=Pressed);(* AND Enable);*)
PressedFlag:=PressedRTrig.Q;

(* Check button enabled *)
IF 	Enable THEN
	(* Button enabled *)
	Button.TextColor:=TextColEnabled;

	(* Check button pressed *)
	IF 	Pressed THEN
		(* Button pressed *)
		Button.BackgroundColor:=ButtBackColor;
	ELSE
		(* Button not pressed *)

		(* Check state on *)
		IF 	StateOn THEN
			(* State on *)
			Button.BackgroundColor:=ButtColOn;
		ELSE
			(* State off *)
			Button.BackgroundColor:=ButtBackColor;
		END_IF

	END_IF
ELSE
	(* Button not enabled *)
	Button.TextColor:=TextColDisabled;
	Button.Pressed:=FALSE;
	(* Check state on *)
	IF 	StateOn THEN
		(* State on *)
		Button.BackgroundColor:=ButtColOn;
	ELSE
		(* State off *)
		Button.BackgroundColor:=ButtColDisabled;
	END_IF

END_IF

(* Additional assigns to visu *)
Button.Enable:=Enable;
Button.Visible:=Visible;

IF 	StateOn THEN
	(* State on *)
	Button.Text:=TextOn;
ELSE
	(* State off *)
	IF 	TextOff<>'' THEN
		Button.Text:=TextOff;
	ELSE
		Button.Text:=TextOn;
	END_IF
END_IF
END_FUNCTION_BLOCK

(* POU zLibrary/_HelpFunctions/FB_Laufschrift_STR255, ST *)
FUNCTION_BLOCK FB_Laufschrift_STR255
VAR_INPUT
	N 					:INT; (* Max output Stringlength *)
	StepWidth			:INT:=1;
	PT					:TIME;
END_VAR
VAR_IN_OUT
	Text 				:STRING(255); (* Original String *)
END_VAR
VAR_OUTPUT
	Display 				:STRING(255); (* Output String *)
END_VAR
VAR
	delay 				:TP;
	TempOutputString	:STRING(255);
	TempInputText		:STRING(255);
	step 				:INT;
END_VAR
(* generate next ticker when delay is low *)
IF 	N < LEN(text) THEN
	IF 	NOT delay.Q THEN
		(* increase step for next tick *)
		TempInputText:=text;

		step := step + StepWidth;

		IF 	step > LEN(TempInputText) THEN
			step := 1;
		END_IF

		(* extract dispay from text *)
		TempOutputString := MID(TempInputText, N, step);

		IF 	LEN(TempOutputString)<N THEN
			TempOutputString:=CONCAT(TempOutputString,TempInputText);
			TempOutputString:=LEFT(TempOutputString,N);
			Display:=TempOutputString;
		ELSE
			Display:=TempOutputString;
		END_IF
		(* set delay timer for next tick *)
		delay(IN := TRUE, PT := PT);
	ELSE
		(* execute delay timer *)
		delay(IN := FALSE);
	END_IF
ELSE
	display := text;
END_IF
END_FUNCTION_BLOCK

(* POU zLibrary/ept/Sprache/ST_Lng, ST *)
PROGRAM ST_Lng (*Pulldownmenue für Sprachumschaltung*)
VAR_OUTPUT
	b_EndChangeLng		: BOOL;
END_VAR
VAR
	b_init				:BOOL:=FALSE;

	b_einblenden		: BOOL;
	fb_Ton_ChangeLng		: TON;
	fb_ton_ausblenden	: TON;
	fb_rTrig_ausblenden	: R_TRIG;

	s_VisuBmpPath		: STRING(255);
	index				: INT;
	i					: INT;
	CURRENTLANGUAGECopy	: STRING(5);

	btn_Language		:ARRAY [0..5] OF sButtonVisuBmp;

END_VAR
fb_Ton_ChangeLng(
	IN:=	ST_ReadXmlLineMsg.b_EndChangeLng AND
			ST_ReadXmlLine.b_EndChangeLng,
	PT:= t#200ms,
	Q=> b_EndChangeLng,
	ET=> );

IF	NOT b_init THEN
	IF	TD.ArtNo <> '' AND
		s_PLC_path <> '' THEN
		b_init:=TRUE;
		CURRENTLANGUAGE:=MP.ST00.Sprache;
		CURRENTLANGUAGECopy:=CURRENTLANGUAGE;
		s_VisuBmpPath:=CONCAT(s_PLC_path, 'bmp\' );
		Btn_Init();
		IF	CURRENTLANGUAGE ='' THEN
			CURRENTLANGUAGE:='DE';
		END_IF
	END_IF
ELSE
	MP.ST00.Sprache := CURRENTLANGUAGE;
END_IF

ST_Lng.btn_Language[ST_Lng.index].BmpPath;
fb_rTrig_ausblenden(CLK:=b_einblenden);
fb_ton_ausblenden(IN:=, PT:=t#5000ms, Q=>);

IF	fb_rTrig_ausblenden.Q THEN
	fb_ton_ausblenden.IN:=NOT fb_ton_ausblenden.IN;
ELSIF
	fb_ton_ausblenden.Q THEN
	fb_ton_ausblenden.IN:=FALSE;
END_IF

IF  b_init THEN
	FOR i := 0 TO 5  BY 1DO
		IF	CURRENTLANGUAGE=btn_Language[i].Text THEN
			index:=i;
			btn_Language[i].innenFarbe:=Color.darkgrey;
		ELSE
			btn_Language[i].innenFarbe:=Color.lightgrey;
		END_IF

		IF	btn_Language[i].tasten THEN
			CURRENTLANGUAGE:=btn_Language[i].Text;
			fb_ton_ausblenden.IN:=FALSE;
		END_IF
	END_FOR
	CURRENTLANGUAGECopy:=CurrentLanguage;
END_IF
END_PROGRAM
ACTION Btn_Init:
(*=====================================================================*)
btn_Language[0].Text:='DE';
btn_Language[1].Text:='EN';
btn_Language[2].Text:='CZ';
btn_Language[3].Text:='';
btn_Language[4].Text:='';
btn_Language[5].Text:='';

FOR i := 0 TO 5  BY 1DO
	btn_Language[i].deaktivieren:=FALSE;
	btn_Language[i].Textfarbe:=Color.black;
	btn_Language[i].BmpPath:=s_VisuBmpPath;

	btn_Language[i].BmpPath:=CONCAT(btn_Language[i].BmpPath,btn_Language[i].Text);
	btn_Language[i].BmpPath:=CONCAT(btn_Language[i].BmpPath,'.bmp');
	IF	btn_Language[i].Text = '' THEN
		btn_Language[i].unsichtbar:= TRUE;
	ELSE
		btn_Language[i].unsichtbar:= FALSE;
	END_IF

END_FOR
END_ACTION

(* POU System/VisuInterface/ModeSelect, ST *)
PROGRAM ModeSelect (*28.JUL 2010, g.baiz (mit korrigiertem iRemoteAutoStart und iRemoteAutoStop) *)

VAR_OUTPUT
	HomePosition				:	BOOL;
	State								: DINT;
	Mode								:	StateMode;	          (*Betriebsarten / mode*)
	BasicManualMode			:	BOOL	:=	FALSE;
	BasicAutoMode				:	BOOL	:=	FALSE;
	QReset							:	BOOL	:=	FALSE;
	GlobalEnable		:	BOOL	:=	TRUE;
	ControlIsOn			: BOOL;
	ManualFirstImp		: BOOL	:=	FALSE;
	StepFirstImp		: BOOL	:=	FALSE;
	AutoFirstImp		: BOOL	:=	FALSE;
	HomePosRunFirstImp	: BOOL	:=	FALSE;
	QProtecKeyNotIn		: BOOL	:=	FALSE;
	QProtecNotBridged	: BOOL	:=	FALSE;
END_VAR
VAR_INPUT
	(* Inputs from SFC's (used from the application programmer) *)
	AskForNoMode			: BOOL;
	AskForManual			: BOOL;
	AskForStepMode			: BOOL;
	AskForStepStop			: BOOL;
	AskForStepStart			: BOOL;
	AskForAutoMode			: BOOL;
	AskForAutoStart			: BOOL;
	AskAutoStartOverHomePosRun : BOOL;
	AskForAutoStop			: BOOL;
	AskForHomePos			: BOOL;
	AskForSpecialMode		: BOOL;
	(**)
	iRemoteAutoStart		: BOOL;
	iRemoteAutoStop			: BOOL;
	(* Inputs from other FB's (used for call in Special) *)
	ControlOn				: BOOL;
	ProtecKeyNotIn			: BOOL;
	ProtecNotBridged		: BOOL;
	EnableFromPrevMach		: BOOL;
	EnableFromNextMach		: BOOL;
	AllDoorsClosed			: BOOL;
	SafetyDoorOk			: BOOL;
	MainValveOk				: BOOL;
	EmergencyOk				: BOOL;
	BusControlState			: DINT;
	UserOK					: BOOL;
	(* Inputs from MainSequences (signal for Sequence-End) *)
	AutoCycleEnd			: BOOL;
	SpecialCycleEnd 		: BOOL;
	HomePosRunEnd			: BOOL;
	DisableManualMode		: BOOL; 	(* Do not show button for manual mode. This can avoid that automatic cycle is interrupted by operator *)
	RunEmptyEnd				: BOOL; 	(*CellIsEmpty*)
	ShowBtnRunEmpty			: BOOL :=TRUE;

	(*Standard-Inputs *)
	sInit					: sModeSelectInit;(* stuct for initializing*)
											(* Initialisierungsstruktur*)
	Enable					: BOOL; 		(* Enables the operations *)
									 		(* Freigabe für Aktion *)
	Reset					: BOOL; 		(* resetting the Objekt *)
											(* Zurücksetzen des Objektes *)
END_VAR

VAR
	BtnManual		: VisuButton;
	BtnStep			: VisuButton;
	BtnStepCycle	: VisuButton;
	BtnAuto			: VisuButton;
	BtnAutoStart	: VisuButton;
	BtnAutoStop		: VisuButton;
	BtnRunEmpty		: VisuButton;
	BtnHomeRun		: VisuButton;
	BtnSpecial		: VisuButton;
	BtnSpecStep		: VisuButton;
	BtnReset		: VisuButton;

	(* Internal Variables *)
	ErrorNo			: DINT;
	ErrorText		: STRING(80);
	InternNextStep	: BOOL;
	InternResetMode	: DINT;
	InternLastMode	: DINT;
	StepToAuto		: BOOL;
	ShowButton		: BOOL;
	HardwareOk		: BOOL;
	ResetFlag		: R_TRIG;
	ton_Reset		: TON;

	HomePositionInfoNo		: DINT;					(* missing to home posistion /  Fehlernummer fehlende Grundstellung *)
 	NoModeFirstImp			: R_TRIG;
	TipInSpecialMode		: BOOL;
END_VAR
VAR_IN_OUT
	sVisu					: sModeSelectVisu;
END_VAR
VAR CONSTANT
	RESET_FOR_MANUAL			: DINT:=1;
	RESET_FOR_STEP				: DINT:=2;
	RESET_FOR_AUTO				: DINT:=3;
	RESET_FOR_MODE_HOME_POS_RUN	: DINT:=4;
END_VAR
(* Manual mode *)
BtnManual(		Button:=sVisu.BtnManual,
				PressedExt:=FALSE ,
				StateOn:= Mode=MODE_MANUAL ,
				TextOn:='Manual',
				TextOff:='Manual',
				);

(* Step  *)
BtnStep(		Button:=sVisu.BtnStep,
				PressedExt:=FALSE ,
				StateOn:= Mode=MODE_STEP OR Mode=MODE_STEP_RUN,
				TextOn:='Step',
				TextOff:='Step',
				);
(* Step cycle *)
BtnStepCycle(	Button:=sVisu.BtnStepCycle,
				PressedExt:=FALSE ,
				StateOn:= gTipImp ,
				TextOn:='StepCycle',
				TextOff:='StepCycle',
				);
(* Auto mode *)
BtnAuto(		Button:=sVisu.BtnAuto,
				PressedExt:=FALSE ,
				StateOn:= (Mode=MODE_AUTO OR Mode=MODE_AUTO_RUN OR Mode=MODE_AUTO_STOP OR Mode=MODE_HOME_POS_RUN),
				TextOn:='Auto',
				TextOff:='Auto',
				);
(* Auto start *)
BtnAutoStart(	Button:=sVisu.BtnAutoStart,
				PressedExt:=FALSE ,
				StateOn:= Mode=MODE_AUTO_RUN,
				TextOn:='AutoStart',
				TextOff:='AutoStart',
				);
(* Auto stop *)
BtnAutoStop(	Button:=sVisu.BtnAutoStop,
				PressedExt:=FALSE ,
				StateOn:= Mode=MODE_AUTO_STOP,
				TextOn:='AutoStop',
				TextOff:='AutoStop',
				);
(* RunEmpty *)
BtnRunEmpty(	Button:=sVisu.BtnRunEmpty,
				PressedExt:=FALSE ,
				StateOn:=gRunEmpty,
				TextOn:='RunEmpty',
				TextOff:='RunEmpty',
				);
(* SpecialMode *)
BtnSpecial(		Button:=sVisu.BtnSpecial,
				PressedExt:=FALSE ,
				StateOn:= Mode=MODE_SPECIAL,
				TextOn:='Special',
				TextOff:='Special',
				);
(* Step in SpecialMode *)
BtnSpecStep(	Button:=sVisu.BtnSpecStep,
				PressedExt:=FALSE ,
				StateOn:= TipInSpecialMode,
				TextOn:= 'StepCycle',
				TextOff:='StepCycle',
				);
(* Home pos run *)
BtnHomeRun(	Button:=sVisu.BtnHomeRun,
				PressedExt:=FALSE ,
				StateOn:= Mode=MODE_HOME_POS_RUN,
				TextOn:='Home',
				TextOff:='Home',
				);
(*Reset *)
BtnReset(		Button:=sVisu.BtnReset,
				PressedExt:=FALSE ,
				StateOn:= gResetAll,
				TextOn:='Reset',
				TextOff:='Reset',
				);
ManualFirstImp:=FALSE;
StepFirstImp:=FALSE;
AutoFirstImp:=FALSE;
HomePosRunFirstImp:=FALSE;

(*###########################################################################*)
(*    Change Visu Picture																															 *)
(*###########################################################################*)
IF 	BtnAutoStart.PressedFlag THEN
	visu.SelectPictureName:='MAIN';
	CurrentVisu:='MAIN';
END_IF

IF 	BtnHomeRun.PressedFlag THEN
	visu.SelectPictureName:='SYSTEM_GST';
	CurrentVisu:='SYSTEM_GST';
END_IF

(*###########################################################################*)
(* Anwahl von Einzel-, Tipp- oder Automatikbetrieb nach Resetimpuls          *)
(* Select mode																															 *)
(*###########################################################################*)
CASE InternResetMode OF
RESET_FOR_MANUAL:
	Mode:=MODE_MANUAL;
	ManualFirstImp:=TRUE;
RESET_FOR_STEP:
	Mode:=MODE_STEP;
	StepFirstImp:=TRUE;
RESET_FOR_AUTO:
	Mode:=MODE_AUTO;
	AutoFirstImp:=TRUE;
RESET_FOR_MODE_HOME_POS_RUN:
	Mode:=MODE_HOME_POS_RUN;
	HomePosRunFirstImp:=TRUE;
END_CASE
InternResetMode:=0;
(*###########################################################################*)
(* 	Einlesen der Tasten der Visualisierung	(CTS-Signal)										 *)
(*	--> Betriebsartenanwahl																									 *)
(*###########################################################################*)

IF 	BtnManual.PressedFlag THEN
	InternResetMode:=RESET_FOR_MANUAL;
END_IF

IF 	BtnStep.PressedFlag THEN
	CASE Mode OF
	MODE_STEP:
		;
	MODE_STEP_RUN,MODE_AUTO_STOP:
		Mode:=MODE_STEP_STOP;
	MODE_AUTO:
		Mode:=MODE_STEP;
	MODE_AUTO_RUN:
		Mode:=MODE_STEP_RUN;
	ELSE
		InternResetMode:=RESET_FOR_STEP;
	END_CASE
END_IF

IF 	BtnStepCycle.PressedFlag THEN
	CASE Mode OF
	MODE_STEP:
		Mode:=MODE_STEP_RUN;
	MODE_STEP_RUN,MODE_STEP_STOP,MODE_SPECIAL:
		InternNextStep:=TRUE;
	END_CASE
ELSE
	InternNextStep:=FALSE;
END_IF

IF 	BtnAuto.PressedFlag THEN
	CASE Mode OF
	MODE_STEP:
		Mode:=MODE_AUTO;
	MODE_STEP_RUN:
		Mode:=MODE_AUTO;
		StepToAuto:=TRUE;
	MODE_STEP_STOP:
		Mode:=MODE_AUTO_STOP;
		StepToAuto:=TRUE;
	MODE_AUTO,MODE_AUTO_RUN,MODE_AUTO_STOP:
		;
	ELSE
		InternResetMode:=RESET_FOR_AUTO;
	END_CASE
END_IF

IF 	BtnAutoStart.PressedFlag OR
	iRemoteAutoStart AND
	(BtnAuto.Visible OR BtnHomeRun.Visible)THEN
	IF 	BtnHomeRun.Visible OR
		Mode<=MODE_MANUAL AND NOT HomePosRunEnd THEN
		Mode:=MODE_HOME_POS_RUN;
  		HomePosRunFirstImp:=TRUE;
		InternLastMode:=MODE_AUTO_RUN;
		iRemoteAutoStart:=FALSE;
	ELSE
		Mode:=MODE_AUTO_RUN;
		StepToAuto:=FALSE;
		iRemoteAutoStart:=FALSE;
	END_IF
END_IF

IF 	BtnAutoStop.PressedFlag OR
 	iRemoteAutoStop AND BtnAutoStop.Visible THEN
	Mode:=MODE_AUTO_STOP;
	iRemoteAutoStop:=FALSE;
END_IF

IF 	BtnRunEmpty.PressedFlag OR gStartRunEmpty THEN
	gRunEmpty:=NOT(gRunEmpty);
END_IF

IF 	BtnHomeRun.PressedFlag THEN
	CASE Mode OF
	MODE_STEP:
		InternLastMode:=MODE_STEP;
		Mode:=MODE_HOME_POS_RUN;
		HomePosRunFirstImp:=TRUE;
	MODE_AUTO:

		InternLastMode:=MODE_AUTO;
		Mode:=MODE_HOME_POS_RUN;
		HomePosRunFirstImp:=TRUE;
	MODE_STEP_STOP:
		InternLastMode:=MODE_STEP;
		InternResetMode:=RESET_FOR_MODE_HOME_POS_RUN;
	MODE_AUTO_STOP:
		InternLastMode:=MODE_AUTO;
		InternResetMode:=RESET_FOR_MODE_HOME_POS_RUN;
	END_CASE
END_IF

IF 	BtnSpecial.PressedFlag THEN
	Mode:=MODE_SPECIAL;
	SpecialCycleEnd:=FALSE;
END_IF

IF 	BtnSpecStep.PressedFlag THEN
	TipInSpecialMode:=NOT(TipInSpecialMode);
END_IF
IF 	Mode<>MODE_SPECIAL THEN
	TipInSpecialMode:=FALSE;
END_IF

(*###########################################################################*)
(* Input-Variables - used from the application programmer										 *)
(* to modifie the mode out of a SFC 											 *)
(*###########################################################################*)
IF 	AskForNoMode THEN
	Mode:=MODE_NON;
	AskForNoMode:=FALSE;
	iRemoteAutoStart:=FALSE;
ELSIF
	AskForManual THEN
	InternResetMode:=RESET_FOR_MANUAL;
	AskForManual:=FALSE;
	iRemoteAutoStart:=FALSE;
ELSIF
	AskForStepMode THEN
	IF Mode<MODE_STEP THEN
		InternResetMode:=RESET_FOR_STEP;
	END_IF
	Mode:=MODE_STEP;
	AskForStepMode:=FALSE;
ELSIF
	AskForStepStart THEN
	IF 	Mode=MODE_STEP AND
		HomePosRunEnd THEN
		Mode:=MODE_STEP_RUN;
	END_IF
	AskForStepStart:=FALSE;
ELSIF
	AskForStepStop THEN
	Mode:=MODE_STEP_STOP;
	AskForStepStop:=FALSE;
ELSIF
	AskForAutoMode THEN
	IF Mode<MODE_STEP THEN
		InternResetMode:=RESET_FOR_AUTO;
	END_IF
	Mode:=MODE_AUTO;
	AskForAutoMode:=FALSE;
ELSIF
	AskForAutoStop THEN
	Mode:=MODE_AUTO_STOP;
	AskForAutoStop:=FALSE;
	iRemoteAutoStart:=FALSE;
ELSIF
	AskForAutoStart THEN
	IF 	Mode=MODE_AUTO AND
		HomePosRunEnd THEN
		Mode:=MODE_AUTO_RUN;
		StepToAuto:=FALSE;
	END_IF
	AskForAutoStart:=FALSE;
ELSIF
	AskForHomePos THEN
	AskForHomePos:=FALSE;
	CASE Mode OF
	MODE_STEP:
		InternLastMode:=MODE_STEP;
		Mode:=MODE_HOME_POS_RUN;
		HomePosRunFirstImp:=TRUE;
	MODE_AUTO:
		InternLastMode:=MODE_AUTO;
		Mode:=MODE_HOME_POS_RUN;
		HomePosRunFirstImp:=TRUE;
	MODE_STEP_STOP:
		InternLastMode:=MODE_STEP;
		InternResetMode:=RESET_FOR_MODE_HOME_POS_RUN;
	MODE_AUTO_STOP:
		InternLastMode:=MODE_AUTO;
		InternResetMode:=RESET_FOR_MODE_HOME_POS_RUN;
	END_CASE
ELSIF
	AskAutoStartOverHomePosRun THEN
	AskAutoStartOverHomePosRun:=FALSE;
	iRemoteAutoStart:=TRUE;
ELSIF
	AskForSpecialMode THEN
	InternResetMode:=RESET_FOR_AUTO;
	Mode:=MODE_SPECIAL;
	AskForSpecialMode:=FALSE;
END_IF

(*###########################################################################*)
(* Check the Key for SafetyDoor-ByPass
when it's put in -> MODE_AUTO_RUN change automaticaly to MODE_AUTO_STOP
when it's turnes -> mode change automaticaly to MODE_MANUAL 					 *)
(*###########################################################################*)
IF 	NOT ProtecKeyNotIn THEN
	CASE Mode OF
	MODE_AUTO_RUN:
		Mode:=MODE_AUTO_STOP;
	END_CASE
END_IF

IF NOT ProtecNotBridged THEN
	CASE Mode OF
	MODE_MANUAL,MODE_NON:
		;
	ELSE
		InternResetMode:=RESET_FOR_MANUAL;
	END_CASE
END_IF

IF	ControlOn AND
	MainValveOk AND
	SafetyDoorOk AND
	EmergencyOk AND
	BusControlState=STATE_OK AND
	UserOK THEN
	HardwareOk:=TRUE;
ELSE
	HardwareOk:=FALSE;
END_IF

IF 	InternResetMode>0 OR
	NOT HardwareOk THEN
	Mode:=MODE_NON;
END_IF

ControlIsOn:=HardwareOk;

(*###########################################################################*)
(* Für Visualisierung: Betriebsarten auf Bit legen													 *)
(*###########################################################################*)
CASE Mode OF
MODE_NON:
	sVisu.ManualOn:=FALSE;
	sVisu.StepOn:=FALSE;
	sVisu.AutoOn:=FALSE;
	sVisu.AutoStartOn:=FALSE;
	sVisu.AutoStopOn:=FALSE;
	sVisu.SpecialOn:=FALSE;
	sVisu.HomePosRunOn:=FALSE;
	sVisu.BasicManualMode:=FALSE;
	sVisu.BasicAutoMode:=FALSE;
	StepToAuto:=FALSE;

MODE_MANUAL:
	sVisu.ManualOn:=TRUE;
	sVisu.StepOn:=FALSE;
	sVisu.AutoOn:=FALSE;
	sVisu.AutoStartOn:=FALSE;
	sVisu.AutoStopOn:=FALSE;
	sVisu.HomePosRunOn:=FALSE;
	sVisu.SpecialOn:=FALSE;
	sVisu.BasicManualMode:=TRUE;
	sVisu.BasicAutoMode:=FALSE;
	StepToAuto:=FALSE;

MODE_STEP,MODE_STEP_RUN:
	sVisu.ManualOn:=FALSE;
	sVisu.StepOn:=TRUE;
	sVisu.AutoOn:=FALSE;
	sVisu.AutoStartOn:=FALSE;
	sVisu.AutoStopOn:=FALSE;
	sVisu.SpecialOn:=FALSE;
	sVisu.HomePosRunOn:=FALSE;
	sVisu.BasicManualMode:=FALSE;
	sVisu.BasicAutoMode:=TRUE;
	IF 	AskForAutoStop OR
		AskForStepStop THEN
		Mode:=MODE_STEP_STOP;
	END_IF

MODE_STEP_STOP:
	IF AutoCycleEnd THEN
		IF AskForAutoStop THEN
			InternResetMode:=RESET_FOR_MANUAL;
			Mode:=MODE_NON;
		ELSIF
			AskForStepStop THEN
			Mode:=MODE_STEP;
		ELSE
			Mode:=MODE_STEP;
		END_IF
	END_IF

MODE_AUTO:
	sVisu.ManualOn:=FALSE;
	sVisu.StepOn:=FALSE;
	sVisu.AutoOn:=TRUE;
	sVisu.AutoStartOn:=FALSE;
	sVisu.AutoStopOn:=FALSE;
	sVisu.HomePosRunOn:=FALSE;
	sVisu.SpecialOn:=TRUE;
	sVisu.BasicManualMode:=FALSE;
	sVisu.BasicAutoMode:=TRUE;

MODE_AUTO_RUN:
	sVisu.AutoStartOn:=TRUE;
	sVisu.AutoStopOn:=FALSE;
	IF AskForAutoStop THEN
		Mode:=MODE_AUTO_STOP;
	END_IF
	StepToAuto:=FALSE;

MODE_AUTO_STOP:
	sVisu.AutoStartOn:=FALSE;
	sVisu.AutoStopOn:=TRUE;
	IF AutoCycleEnd THEN
		IF NOT sInit.RemoteAutoStopToManual THEN
			Mode:=MODE_AUTO;
		ELSE
			Mode:=MODE_MANUAL;
		END_IF
	END_IF

MODE_HOME_POS_RUN:
	sVisu.ManualOn:=FALSE;
	sVisu.HomePosRunOn:=TRUE;
	sVisu.BasicManualMode:=FALSE;
	sVisu.BasicAutoMode:=TRUE;
	IF 	HomePosRunEnd THEN
		CASE InternLastMode OF
		MODE_STEP:
			Mode:=MODE_STEP;
		MODE_AUTO:
			Mode:=MODE_AUTO;
		MODE_AUTO_RUN: (*is used as next Mode*)
			Mode:=MODE_AUTO_RUN;
		ELSE
			Mode:=MODE_NON;
		END_CASE
	END_IF

MODE_SPECIAL:
	sVisu.SpecialOn:=TRUE;
	IF SpecialCycleEnd THEN
		Mode:=MODE_AUTO;
	END_IF
END_CASE
sVisu.RunEmptyOn:=gRunEmpty;

(*###########################################################################*)
(* Leerfahren zurücksetzen*)
(*###########################################################################*)
IF 	gRunEmpty AND
	RunEmptyEnd AND
	Mode=MODE_AUTO_RUN THEN
	gRunEmpty:=FALSE;
	RunEmptyEnd:=FALSE;
	Mode:=MODE_AUTO_STOP;
END_IF
IF 	gRunEmpty AND
	Mode<=MODE_MANUAL THEN
	gRunEmpty:=FALSE;
END_IF

(*###########################################################################*)
(* State des Betriebsartenbausteins zuweisen*)
(*###########################################################################*)
IF 	gInitOk AND
	gSetupOk THEN
	CASE Mode OF
		MODE_NON:
			IF	NOT ControlOn THEN
				State:=-2;						(* Steuerung einschalten!*)
			ELSE
				State:=-3;						(*Betriebsart anwählen!  *)
			END_IF
			(* SafetyDoor *)
			IF	NOT SafetyDoorOk THEN
				State:=-1;						(* Türe ist auf! *)
			END_IF
			(* MainValve *)
			IF NOT MainValveOk THEN
				State:=-7;						(* Hauptluft darf nicht ein sein!*)
			END_IF
			(* Emergency Stop*)
			IF NOT EmergencyOK THEN
				State:=-1;						(* Not-Aus betätigt! *)
			END_IF
			(* BusControl *)
			IF 	BusControlState<>STATE_OK THEN
				State:=-6;						(* Bus steht! *)
			END_IF
		MODE_MANUAL:
				State:=1;						(* Einzelbetrieb aktiv *)
		MODE_STEP:
			IF HomePosRunEnd THEN
				State:=2;							(* Tippbetrieb vorgewählt *)
			ELSE
				State:=-4;							(* Grundstellung fehlt *)
			END_IF
		MODE_STEP_RUN:
			State:=4;								(* Tippbetrieb läuft *)
		MODE_STEP_STOP:
			State:=10;								(* Tippbetrieb in letzten Zyklus *)
		MODE_AUTO:
			IF HomePosRunEnd THEN
				State:=3;							(* Automatikbetrieb vorgewählt *)
			ELSE
				State:=-4;							(* Grundstellung fehlt *)
			END_IF
		MODE_AUTO_RUN:
			State:=5;								(* Automatikbetrieb läuft *)
		MODE_AUTO_STOP:
			State:=6;								(* Automatikbetrieb im letzen Zyklus *)
		MODE_HOME_POS_RUN:
			State:=7;								(* Grundstellung wird angefahren *)
		MODE_SPECIAL:
			State:=8;								(* Spezialbetrieb läuft *)
	ELSE
			State:=0;								(* nicht definierter Status *)
	END_CASE
	IF 	NOT ProtecKeyNotIn THEN
		State:=16;									(* Schlüsselschalter ist gesteckt *)
	END_IF
	IF 	NOT ProtecNotBridged THEN
		State:=17;									(* Schutz ist überbrückt *)
	END_IF

ELSE
	State:=0;										(* nicht definierter Status *)
END_IF

(* copy input to output parameter *)
QProtecKeyNotIn		:= ProtecKeyNotIn;
QProtecNotBridged	:= ProtecNotBridged;
(*#################### Ende State zuweisen #################################*)
ErrorNo:=0;
ErrorText:='';
(*##########################################################################*)
(* Check home position																											*)
(* Pruefen der Grundstellung																								*)
(*##########################################################################*)
IF	NOT ProtecNotBridged THEN
	HomePositionInfoNo:=11;
ELSIF
	NOT ProtecKeyNotIn THEN
	HomePositionInfoNo:=10;
ELSE
	HomePositionInfoNo:=State_OK;
END_IF
(* Generating home position*)
(* Zuweisung der Grundstellung*)
IF 	HomePositionInfoNo=State_OK THEN
	HomePosition:=TRUE;
ELSE
	HomePosition:=FALSE;
END_IF
(* Objekt-Grundstellung verknüpfen mit GesamtGrundstellung *)
(* object-homeposition concat with mainhomeposition *)
gHomeOk:=gHomeOk AND HomePosition;

(*###########################################################################*)
(* Zuweisungen für Anzeigen am Display -> in sVisu. ...        															 *)
(*###########################################################################*)
(* buttons anzeigen *)
ShowButton:=HardwareOk;

BtnReset.Enable		:= TRUE;
BtnReset.Visible			:= Mode<=MODE_MANUAL;

BtnManual.Enable		:= ShowButton AND (DisableManualMode=FALSE OR Mode<=MODE_MANUAL) AND NOT(sInit.HideManualButton);
BtnManual.Visible		:= BtnManual.Enable;

BtnStep.Enable			:= ProtecNotBridged AND MainValveOk AND SafetyDoorOk AND NOT(Mode=MODE_SPECIAL) AND ShowButton;
BtnStep.Visible			:= BtnStep.Enable;

BtnStepCycle.Enable	:= (Mode=MODE_STEP OR Mode=MODE_STEP_RUN OR Mode=MODE_STEP_STOP OR TipInSpecialMode) AND NOT(BtnHomeRun.Visible) AND ShowButton AND NOT(sInit.HideNextStepButton);
BtnStepCycle.Visible		:= BtnStepCycle.Enable;

BtnAuto.Enable			:= ProtecNotBridged AND MainValveOk AND SafetyDoorOk AND NOT(Mode=MODE_SPECIAL) AND ShowButton;
BtnAuto.Visible			:= BtnAuto.Enable;

BtnAutoStart.Enable		:= (sVisu.AutoStartOn OR sVisu.AutoOn) AND
							Mode<>MODE_SPECIAL AND
							Mode<>MODE_AUTO_STOP AND
							(sInit.EnableQuickAutoStart OR NOT BtnHomeRun.Visible) AND
							ShowButton;
BtnAutoStart.Visible		:= BtnAutoStart.Enable;

BtnAutoStop.Enable		:= (Mode=MODE_AUTO_RUN OR Mode=MODE_AUTO_STOP) AND ShowButton;
BtnAutoStop.Visible		:= BtnAutoStop.Enable;

BtnRunEmpty.Enable	:= (Mode=MODE_AUTO_RUN OR Mode=MODE_AUTO_STOP OR Mode=MODE_AUTO) AND
						ShowBtnRunEmpty AND
						ShowButton AND
						NOT gRunEmpty;
BtnRunEmpty.Visible		:= Mode>MODE_MANUAL AND NOT BtnHomeRun.Visible;

BtnHomeRun.Enable	:= (	(Mode=MODE_AUTO OR Mode=MODE_STEP) AND
							NOT(HomePosRunEnd) OR
							Mode=MODE_HOME_POS_RUN OR
							Mode=MODE_AUTO_STOP OR
							Mode=MODE_STEP_STOP		) AND
							NOT(StepToAuto) AND
							ShowButton;
BtnHomeRun.Visible		:= BtnHomeRun.Enable;

BtnSpecial.Enable		:=  (Mode=MODE_AUTO AND NOT(BtnHomeRun.Visible) AND AutoCycleEnd AND HomePosRunEnd OR Mode=MODE_SPECIAL) AND ShowButton;
BtnSpecial.Visible		:= BtnSpecial.Enable;

BtnSpecStep.Enable		:= Mode=MODE_SPECIAL AND ShowButton;
BtnSpecStep.Visible		:=	BtnSpecStep.Enable;

(* interne Variablen *)
sVisu.State				:= State;
sVisu.HomePositionOk	:= HomePosRunEnd;
sVisu.HomePositionInfoNo:= HomePositionInfoNo;

(*###########################################################################*)
(* Zuweisen der Output-Variablen	        															 *)
(*###########################################################################*)
BasicManualMode	:= sVisu.BasicManualMode;
BasicAutoMode		:= sVisu.BasicAutoMode;
(*---------------------------------------------------------------------------
NextStep for StepMode and SemiAuotomaticMode 
Schrittweiterschaltung bei Tipp- und Teilautomatikbetrieb
  ---------------------------------------------------------------------------*)
CASE Mode OF
MODE_AUTO_RUN,MODE_AUTO_STOP,MODE_HOME_POS_RUN,MODE_SPECIAL:
	IF 	TipInSpecialMode THEN
		gTipImp:=InternNextStep;
	ELSE
		gTipImp:=TRUE;
	END_IF
ELSE
	gTipImp:=InternNextStep;
END_CASE
(*---------------------------------------------------------------------------
Reset for movements and functions 
Reset der Bewegungen und Funktionen
  ---------------------------------------------------------------------------*)

NoModeFirstImp(CLK:= (Mode=MODE_NON) );
ResetFlag(CLK:=NoModeFirstImp.Q OR BtnReset.Pressed);
QReset:=ResetFlag.Q;
ton_Reset(PT:= T#500ms, Q=>);

(*Reset für Tampondrucker*)
IF 	BtnReset.Pressed AND NOT ton_Reset.Q THEN
	ST00_72_K7.SetSignalHigh:=TRUE;
  	ton_Reset.IN := TRUE;
ELSIF
	ton_Reset.Q THEN
	ST00_72_K7.SetSignalLow:=TRUE;
	ton_Reset.IN := FALSE;
END_IF

(*---------------------------------------------------------------------------
Stop and Reset all sequences with : SFCInit-Flag 
Alle Schrittketten stoppen und zurücksetzen mit : SFCInit-Flag
  ---------------------------------------------------------------------------*)
CASE Mode OF
MODE_MANUAL,MODE_STEP_RUN,MODE_STEP_STOP,MODE_AUTO_RUN,MODE_AUTO_STOP,MODE_HOME_POS_RUN,MODE_SPECIAL:
	SFCInit:=FALSE;
MODE_AUTO:
	IF 	StepToAuto THEN
		SFCInit:=FALSE;
	ELSE
		SFCInit:=TRUE;
	END_IF
ELSE
	SFCInit:=TRUE;
END_CASE

(*---------------------------------------------------------------------------
Break to all sequences with : SFCPause-Flag 
Alle Schrittketten unterbrechen mit : SFCPause-Flag
  ---------------------------------------------------------------------------*)
IF 	NOT EnableFromPrevMach AND
	ProtecNotBridged THEN
	GlobalEnable:=FALSE;
	SFCTipMode:=TRUE;
	ErrorNo:=10;
	ErrorText:='Break from Previous Machine';
ELSIF
	NOT EnableFromNextMach AND
	ProtecNotBridged THEN
	GlobalEnable:=FALSE;
	SFCTipMode:=TRUE;
	ErrorNo:=11;
	ErrorText:='Break from Next Machine';
ELSE
	GlobalEnable:=TRUE;
	SFCTipMode:=FALSE;
END_IF

(*$$$$$$$$$$$$$$$$$$$$$$$$$$$$$$$$$$$$$$$$$$$$$$$$$$$$$$$$$$$$$$$$$$$$$$$$$$$
ErrorHandler
$$$$$$$$$$$$$$$$$$$$$$$$$$$$$$$$$$$$$$$$$$$$$$$$$$$$$$$$$$$$$$$$$$$$$$$$$$$*)
IF ErrorNo<>0 THEN
	;
END_IF

(*$$$$$$$$$$$$$$$$$$$$$$$$$$$$$$$$$$$$$$$$$$$$$$$$$$$$$$$$$$$$$$$$$$$$$$$$$$$
Reset of input variables.
$$$$$$$$$$$$$$$$$$$$$$$$$$$$$$$$$$$$$$$$$$$$$$$$$$$$$$$$$$$$$$$$$$$$$$$$$$$*)
DisableManualMode:=FALSE;
END_PROGRAM

(* POU Stations/ST_00/ST00_SFCs/_SpecialModeSFCs/SpecialMode03, SFC *)
PROGRAM SpecialMode03 (*Used for: Beschriften von Nest 1 - Einlegen nach Laser (Station 6) *)
VAR_OUTPUT
	SFCCurrentPOU		: STRING:='SpecialMode03';
	SFCCurrentStep	: STRING:='';
	SFCTime					:	DINT;
  State   				:	DINT;
  Result  				:	DINT;
END_VAR
VAR_INPUT
	Start						:	BOOL;
END_VAR
VAR
	MsgOK				:	BOOL;
	MsgCancel		:	BOOL;
	SFCRun					:	BOOL;
	SFCTimeStart		:	TIME;

	(* Userdefinded area *)

END_VAR
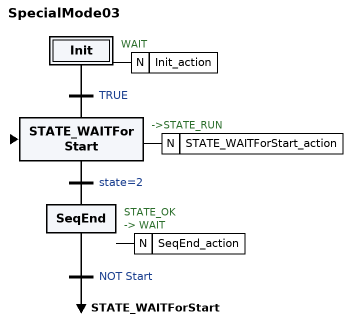
INITIAL_STEP Init: (* WAIT *)
	Init_action(N);
END_STEP
TRANSITION FROM Init TO STATE_WAITForStart := TRUE;
END_TRANSITION
STEP STATE_WAITForStart: (* ->STATE_RUN *)
	STATE_WAITForStart_action(N);
END_STEP
TRANSITION FROM STATE_WAITForStart TO SeqEnd := state=2;
END_TRANSITION
STEP SeqEnd: (* STATE_OK / -> WAIT *)
	SeqEnd_action(N);
END_STEP
TRANSITION FROM SeqEnd TO STATE_WAITForStart := NOT Start;
END_TRANSITION

ACTION Init_action:
Start:=FALSE;
State:=STATE_WAIT;
END_ACTION

ACTION STATE_WAITForStart_action:
IF Start=TRUE
THEN
	State:=STATE_RUN;
	Result:=RESULT_NON;
	SFCTimeStart:=TIME();
(*ELSE*)
END_IF
END_ACTION

ACTION SeqEnd_action:
IF 	State=STATE_RUN THEN
	SFCTime:=TIME_TO_DINT(TIME()-SFCTimeStart);
	State:=STATE_OK;
END_IF

IF 	NOT Start THEN
	State:=STATE_WAIT;
END_IF
END_ACTION
END_PROGRAM

(* POU Stations/ST_00/ST00_SFCs/CheckSFCInInit, ST *)
PROGRAM CheckSFCInInit

VAR_OUTPUT

  AllSeqInInit	:	BOOL;

END_VAR
 AllSeqInInit:=
	ST03_Main.State=STATE_WAIT AND
	ST02_Main.State=STATE_WAIT AND
	(ST08_Process.State=STATE_WAIT OR ST08_Process.State=STATE_OK ) AND
	ST08_Palletizing.State=STATE_WAIT AND
	ST08_Depalletizing.State=STATE_WAIT
;
END_PROGRAM

(* POU Stations/ST_03_Ruestsaetze/ST_03_SFCs/ST03_Main, SFC *)
PROGRAM ST03_Main

VAR_OUTPUT
	SFCCurrentPOU			: STRING:='ST03_Main';
	SFCCurrentStep			: STRING:='';
	FB_CurrentStepHistorie	: FB_CurrentStepHistorie;
	SFCTime					: DINT;
	State   				: StateObject	:= STATE_WAIT;

	Nest10Locked			: BOOL;
	Nest10Done				: BOOL;
	IstPosHelp				: LREAL;
END_VAR
VAR_INPUT
	RunEmpty				: BOOL;
	TestPartsRemove			: BOOL;
	Result 					: DINT;
END_VAR
VAR
	MsgOK					: BOOL;
	MsgCancel				: BOOL;
	SFCRun					: BOOL;
	SFCTimeStart			: TIME;
	Delay					: TON;
	Error					: ErrorStruct;
	(* Userdefinded area *)
	AnzahlTeile   			: DINT;
	PutIdx					: DINT;
	Nest_Empty      		: BOOL;
	kein_Teil_NOK			: BOOL;
	CTR						: DINT;
	CTR2					: DINT;
	Result_help				: DINT;
END_VAR
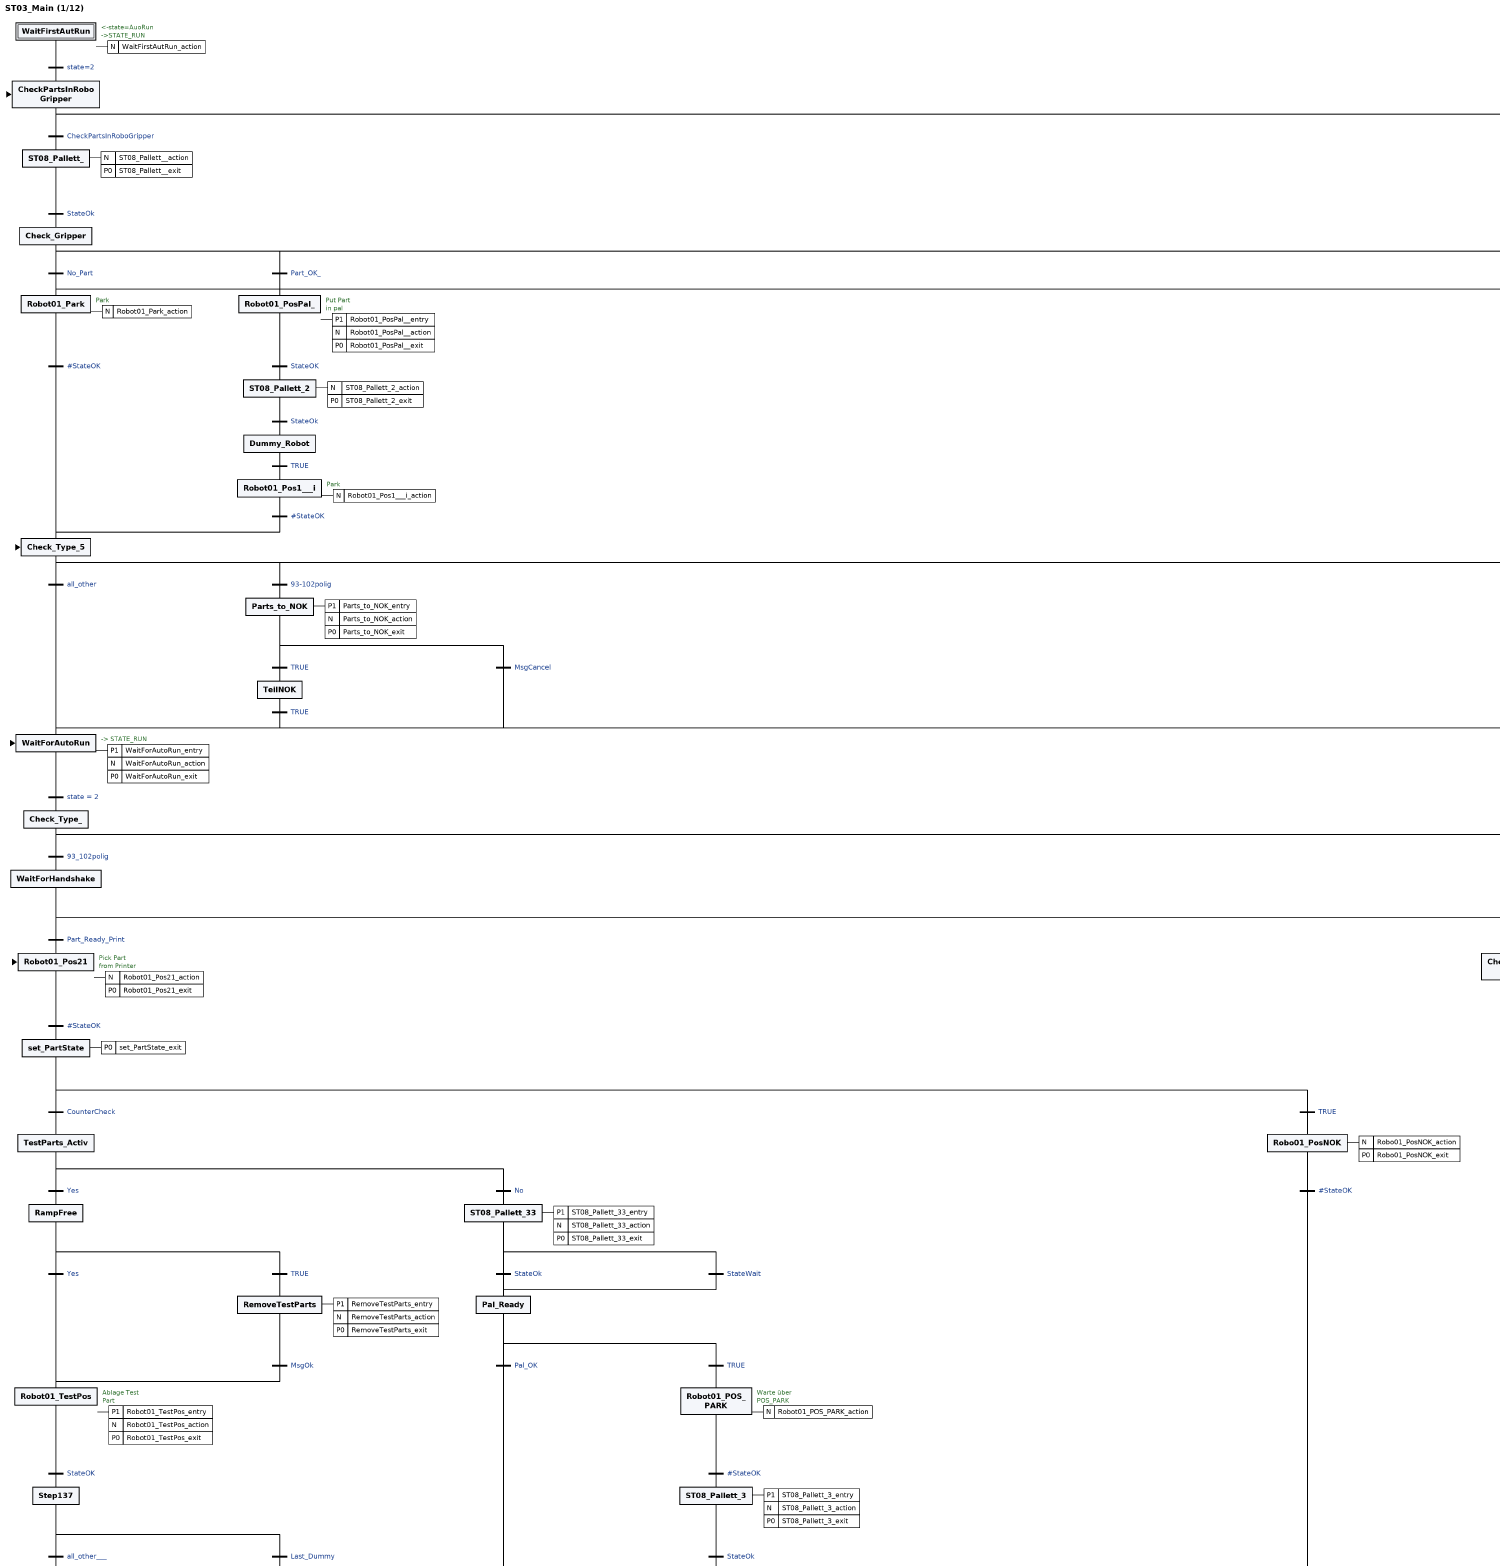
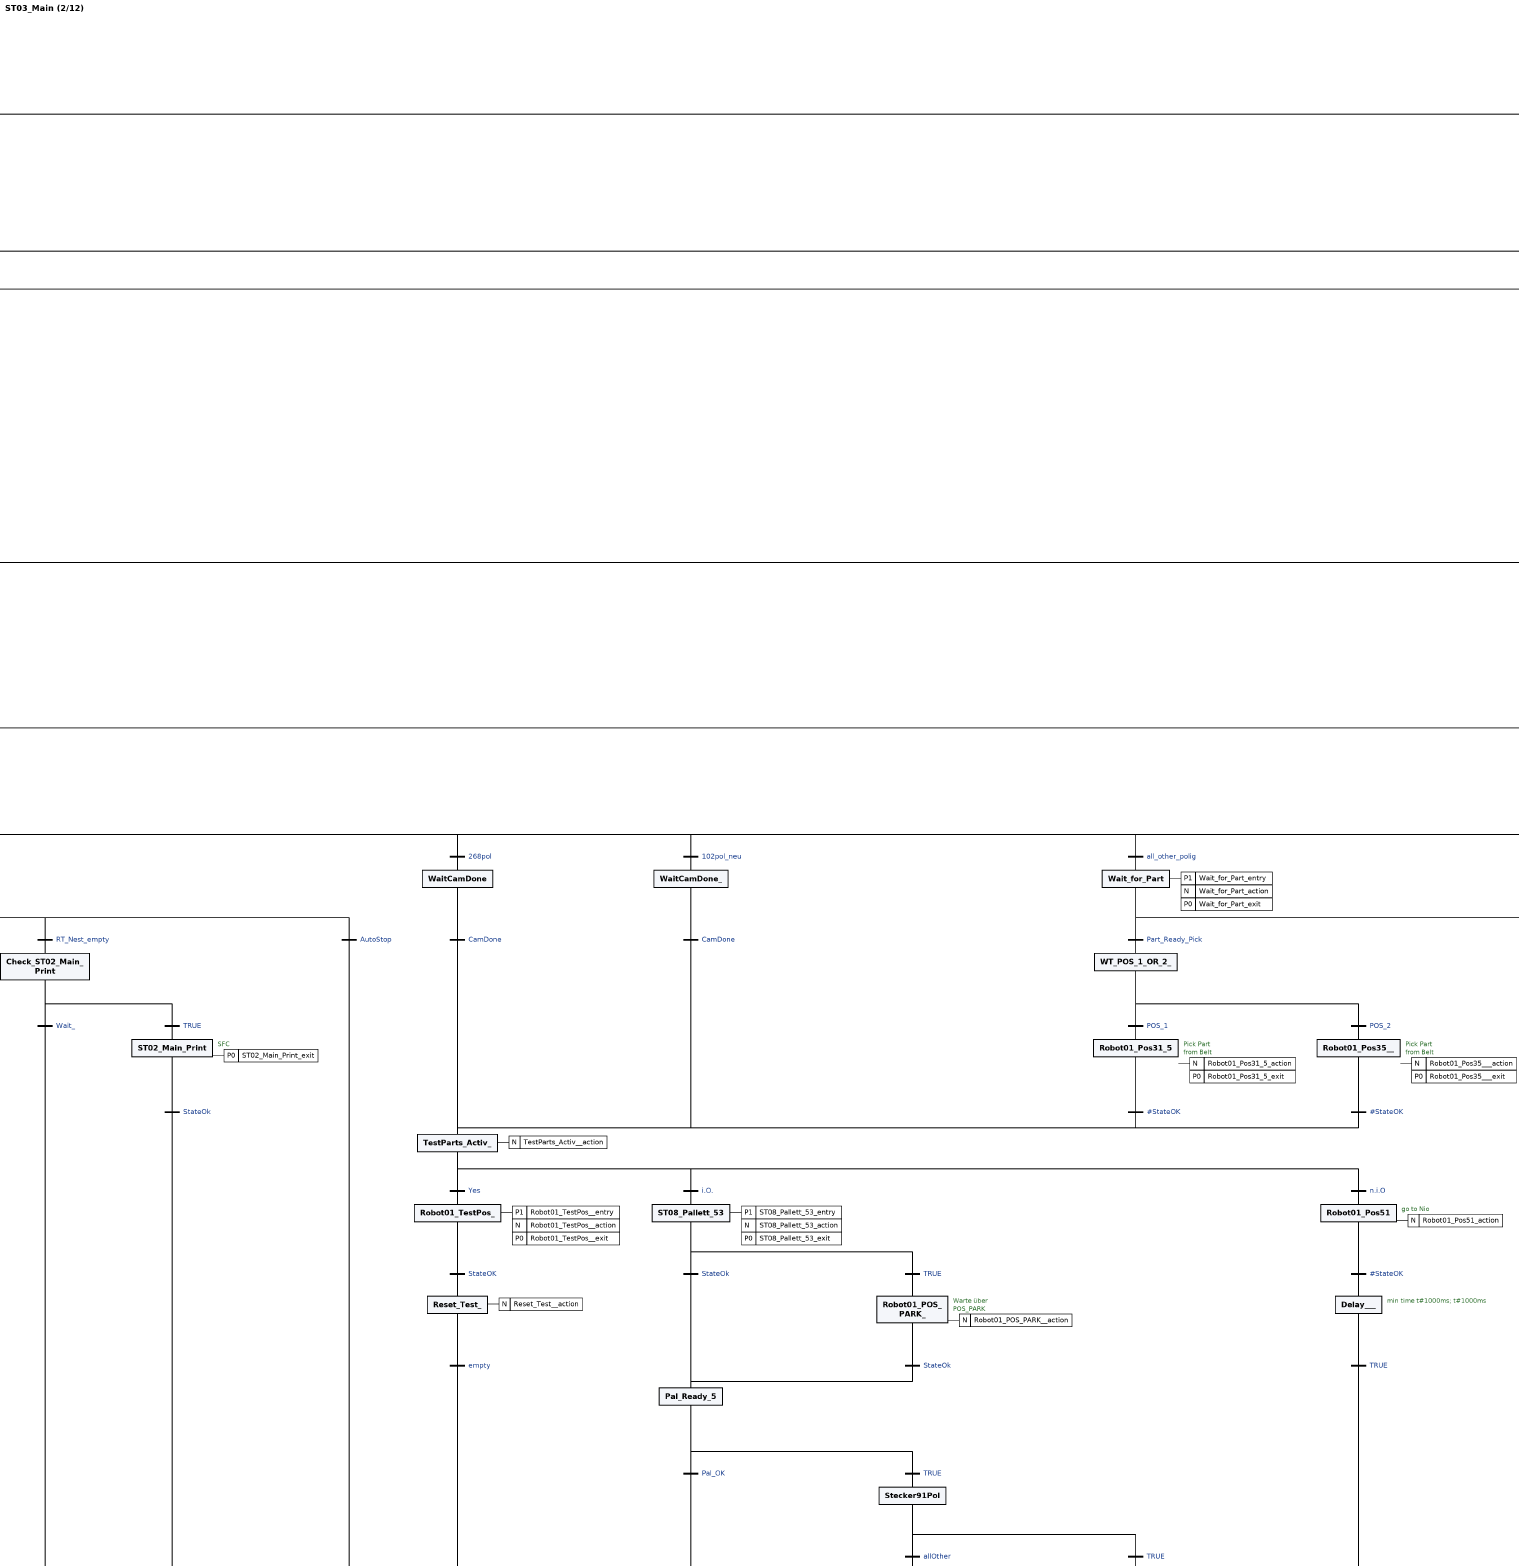
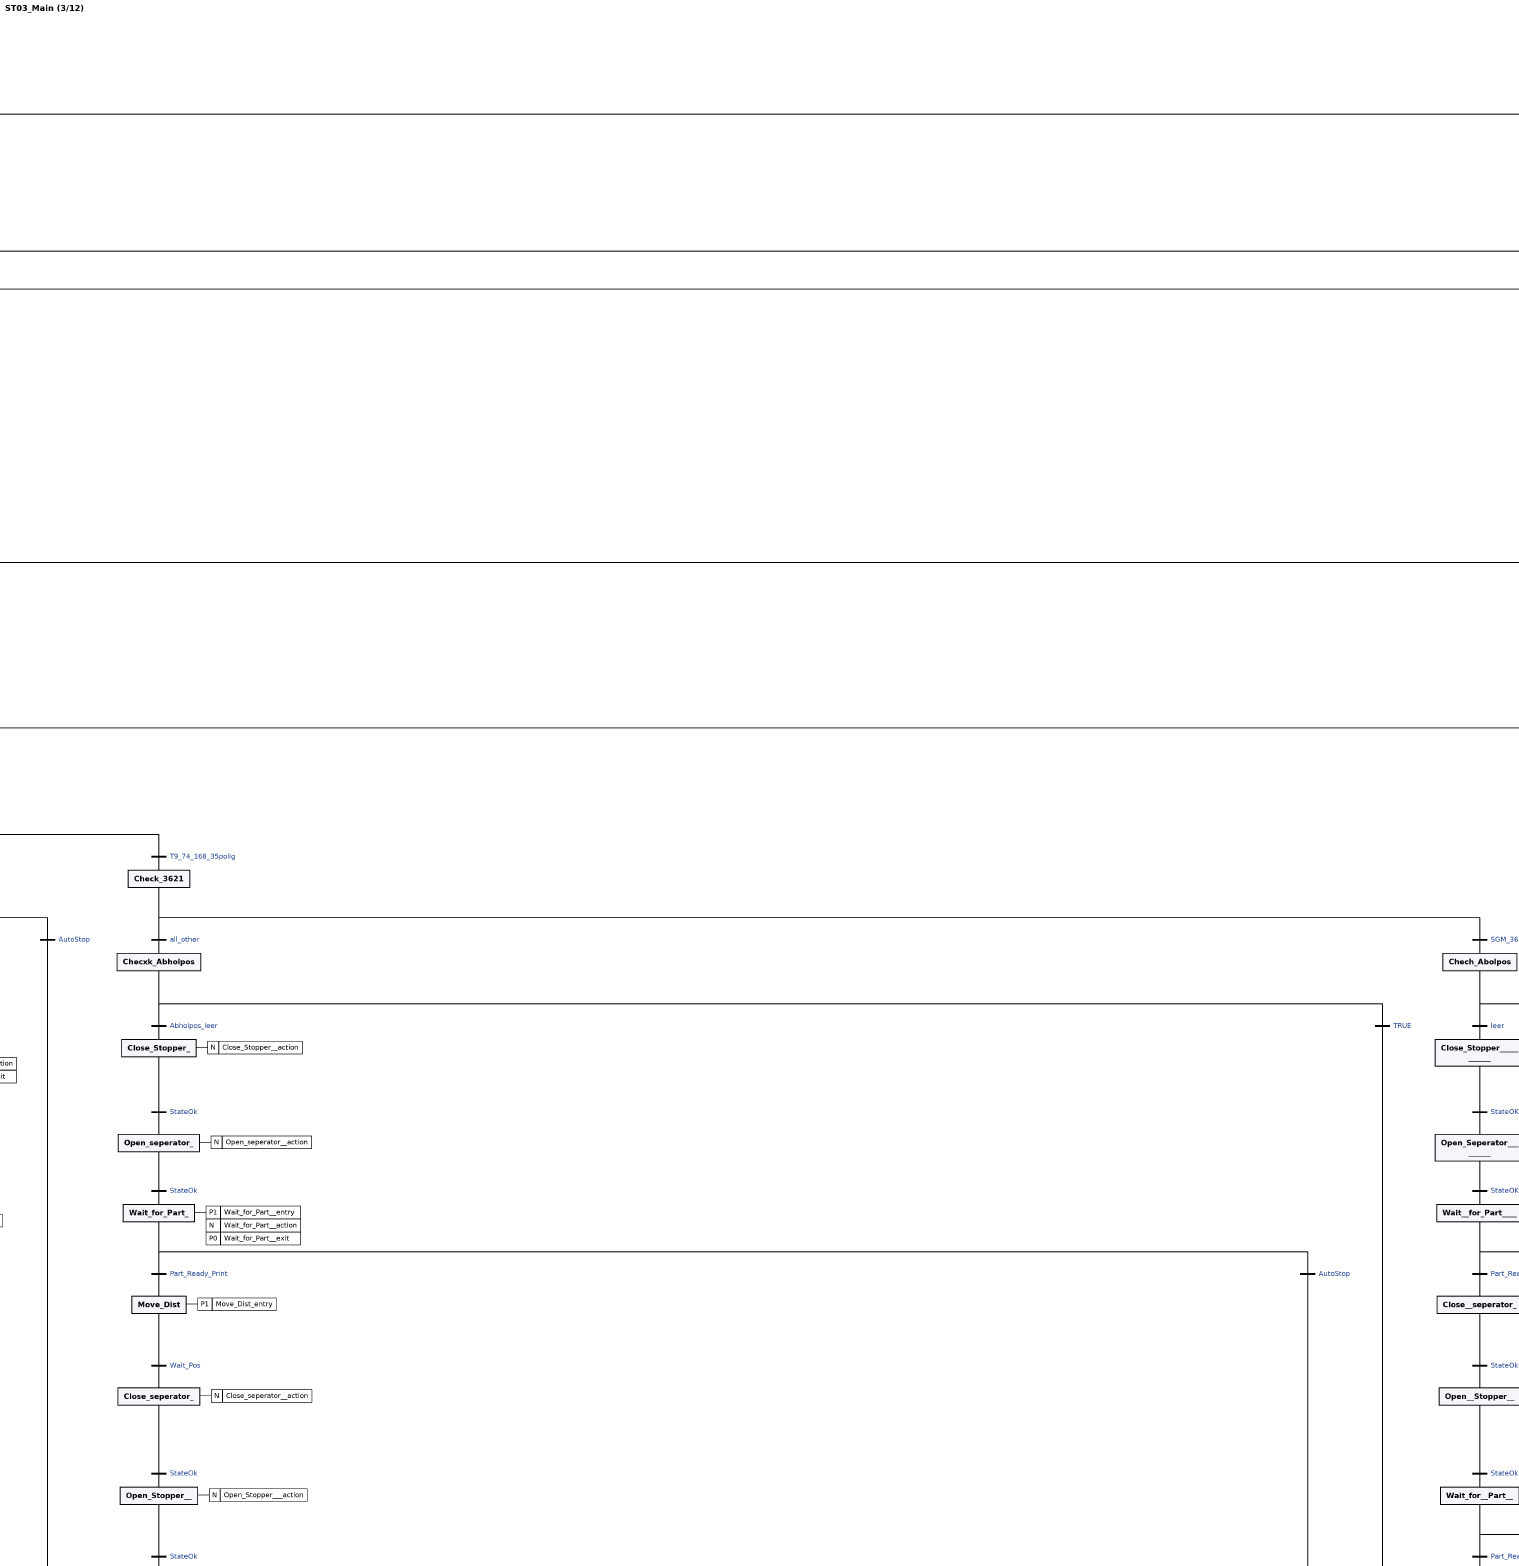
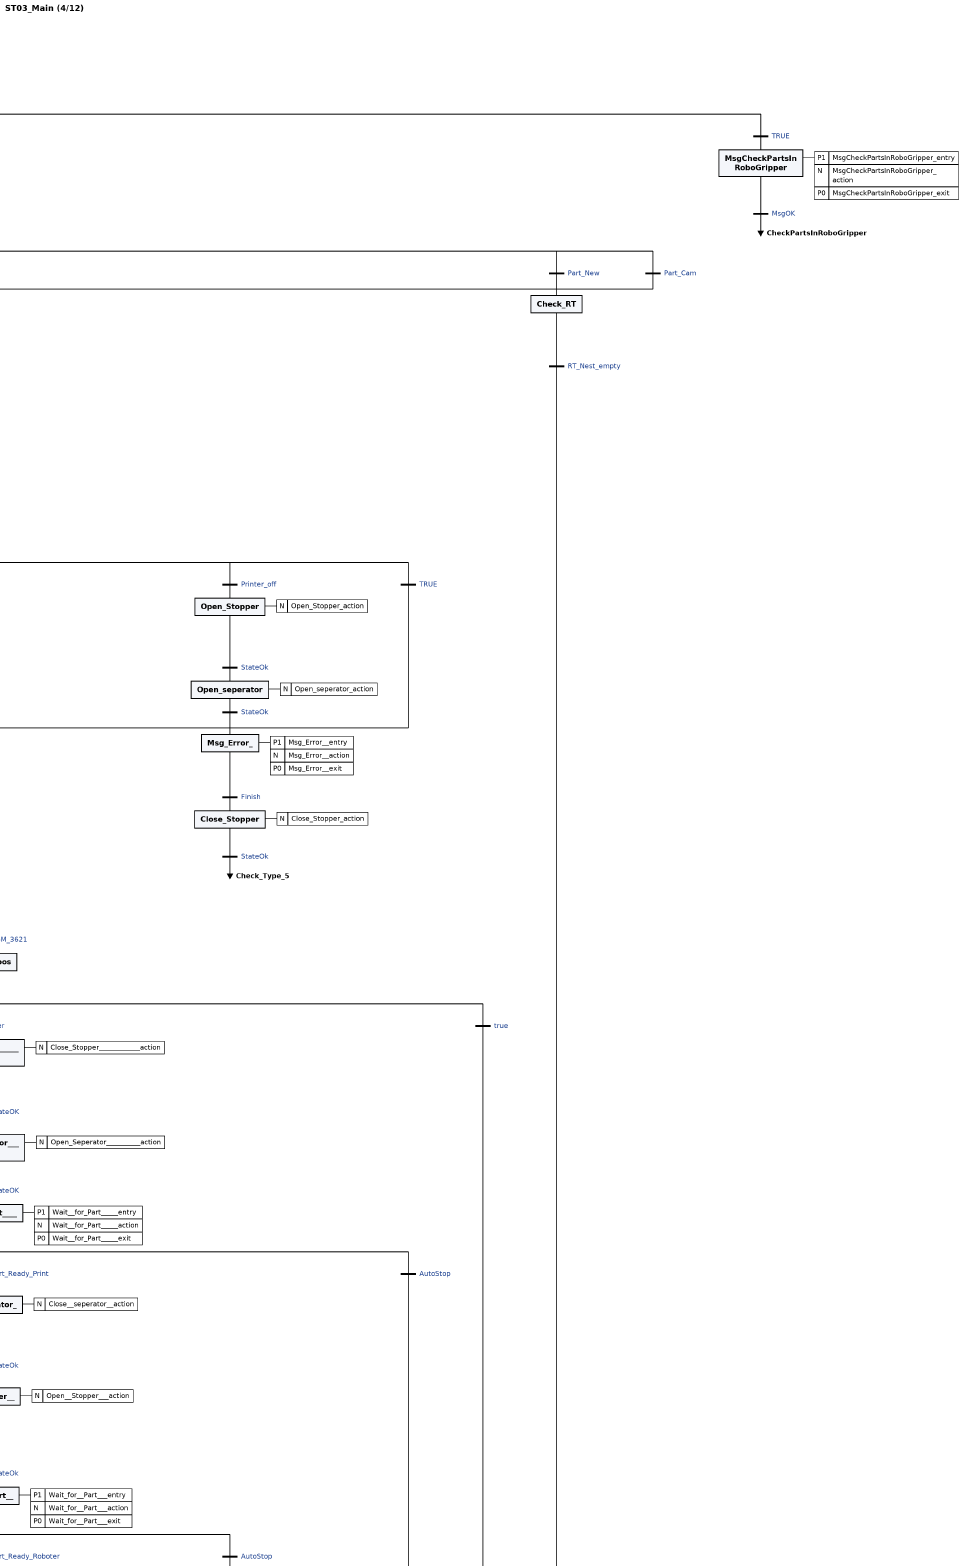
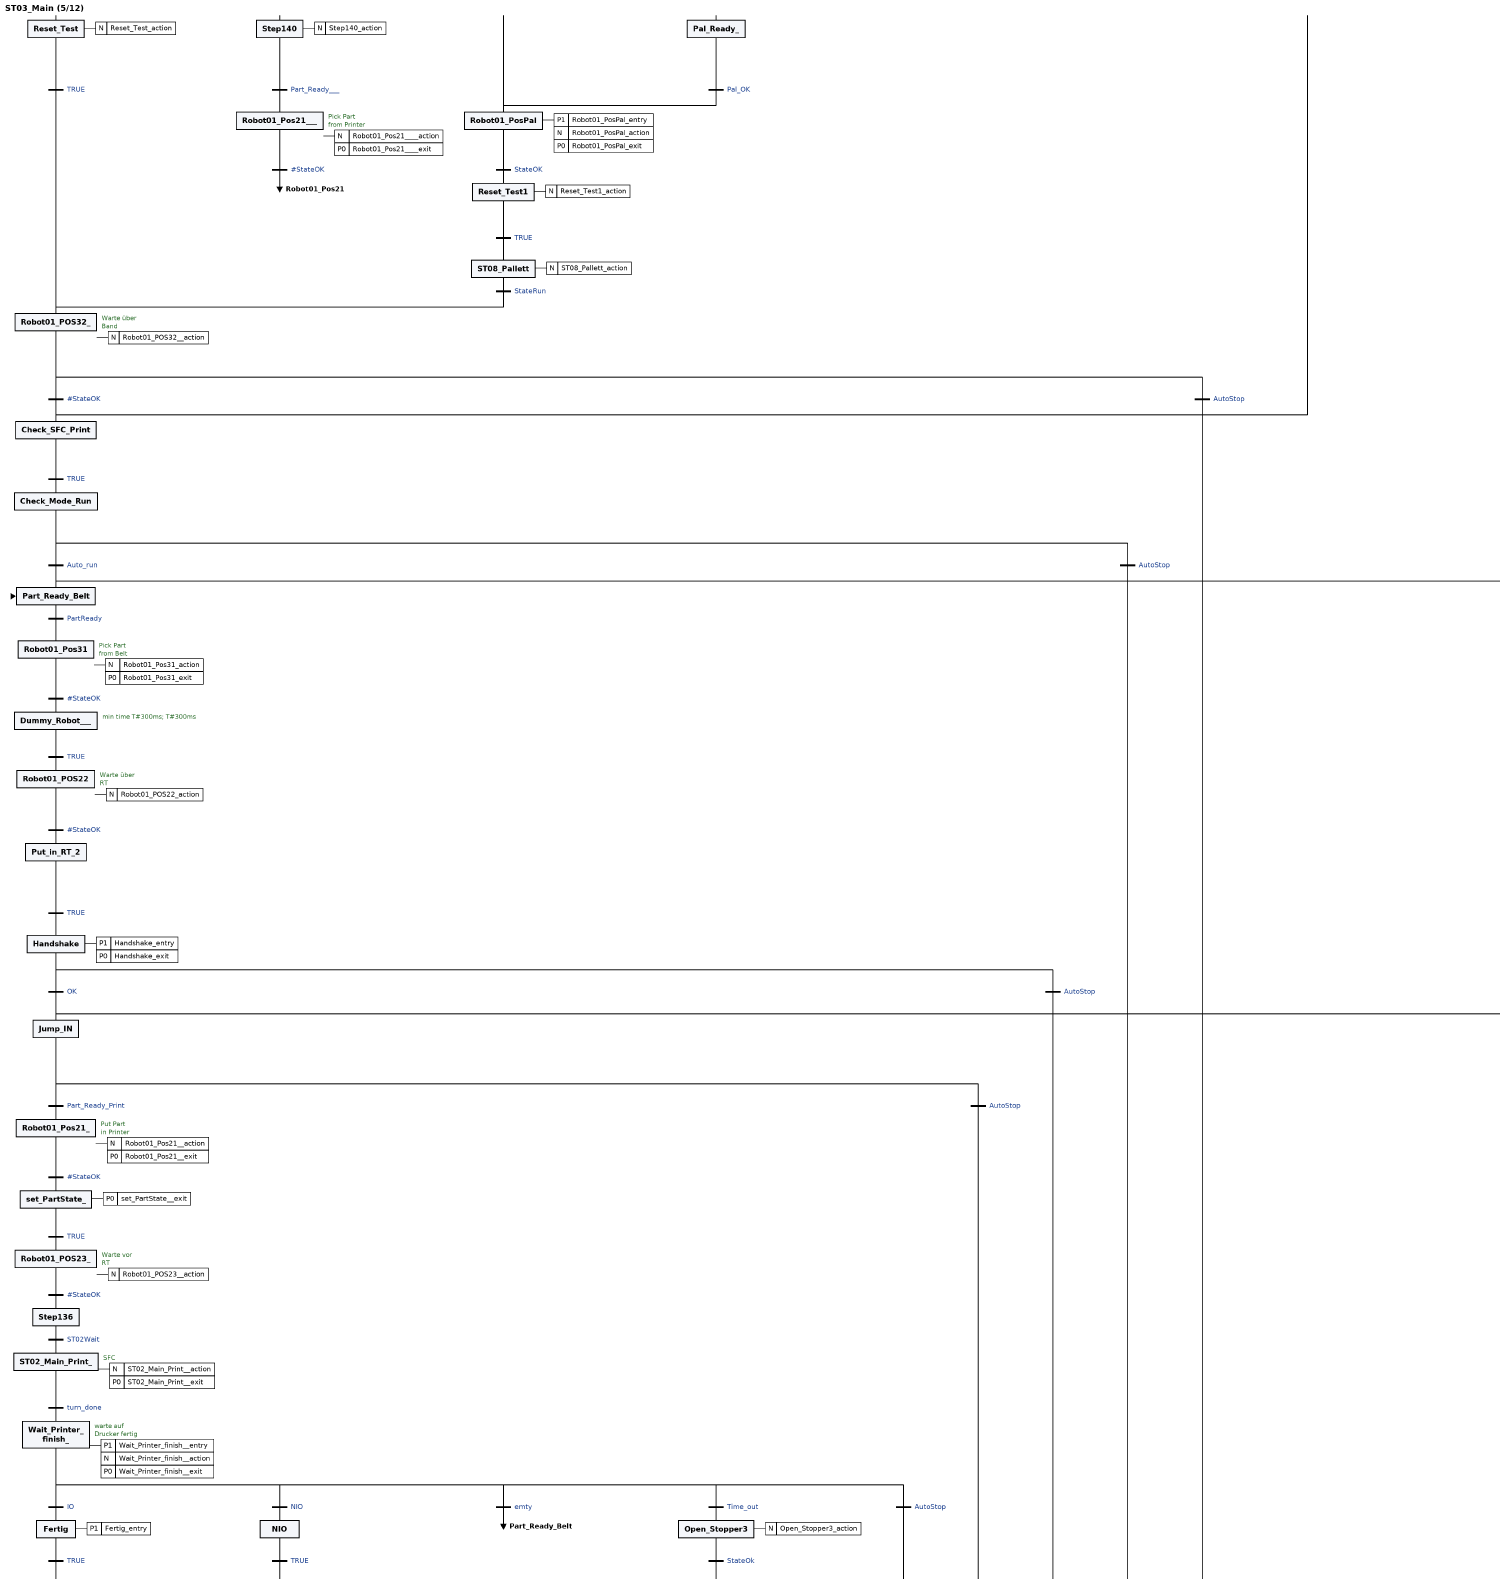
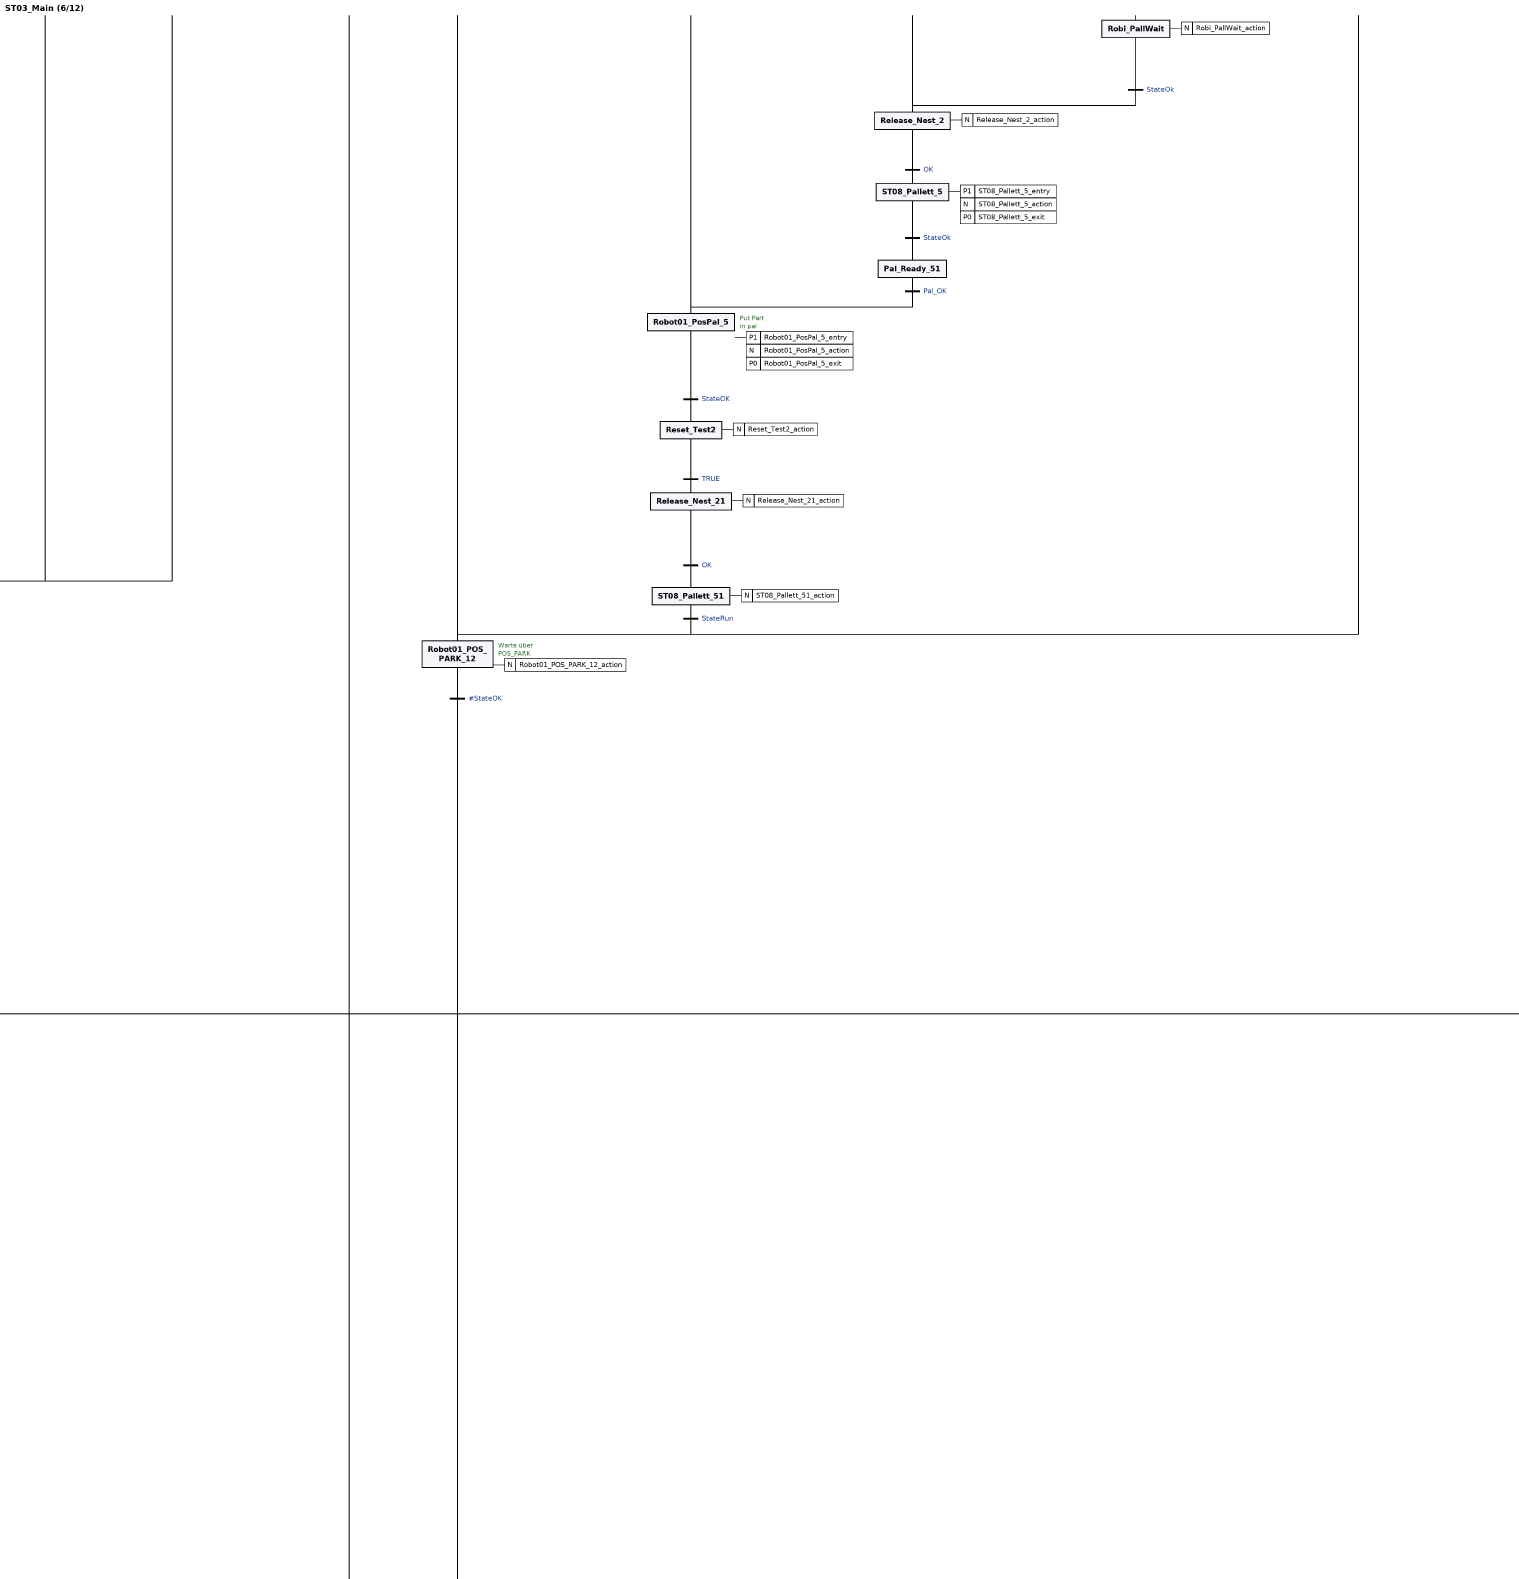
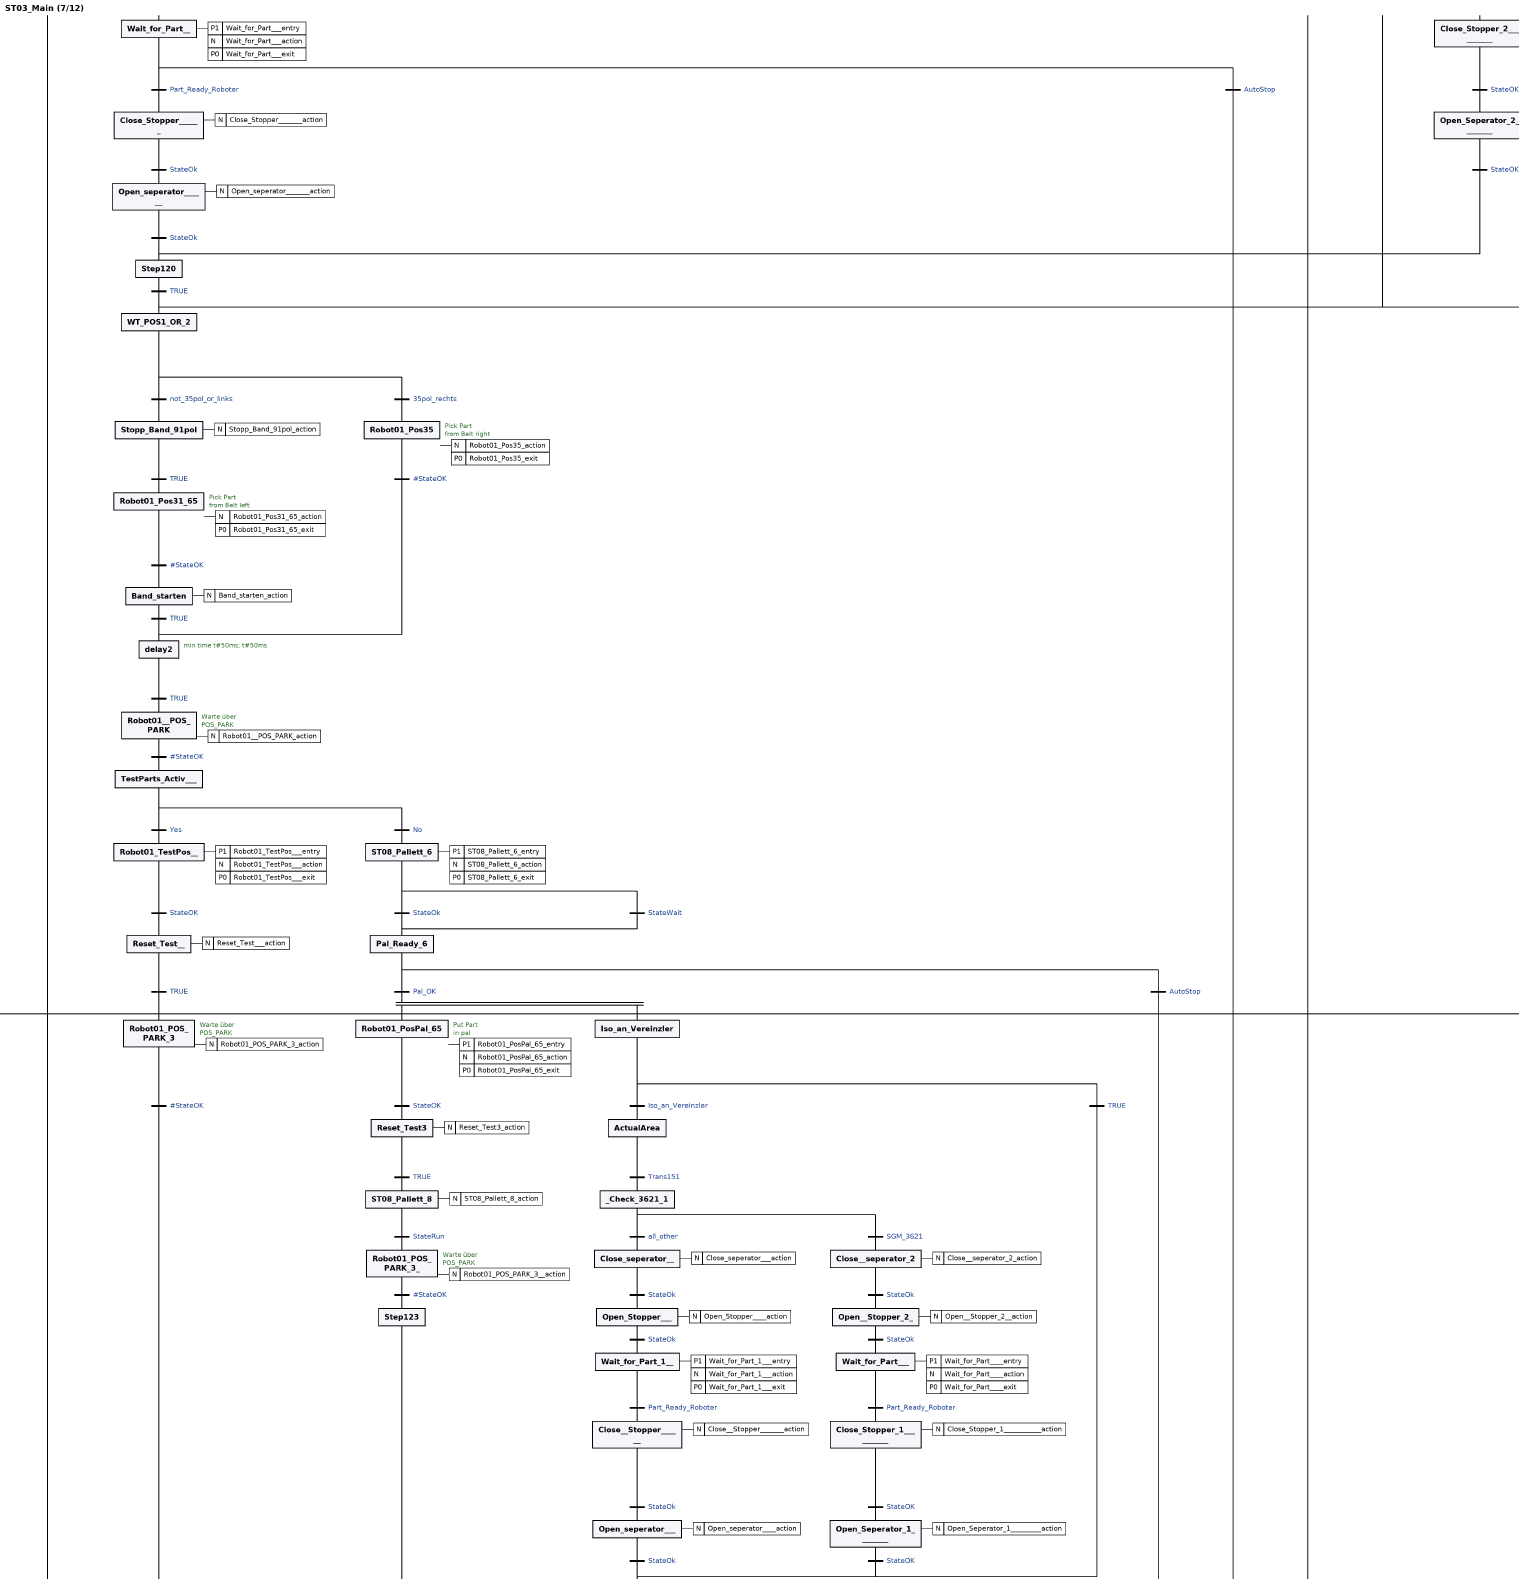
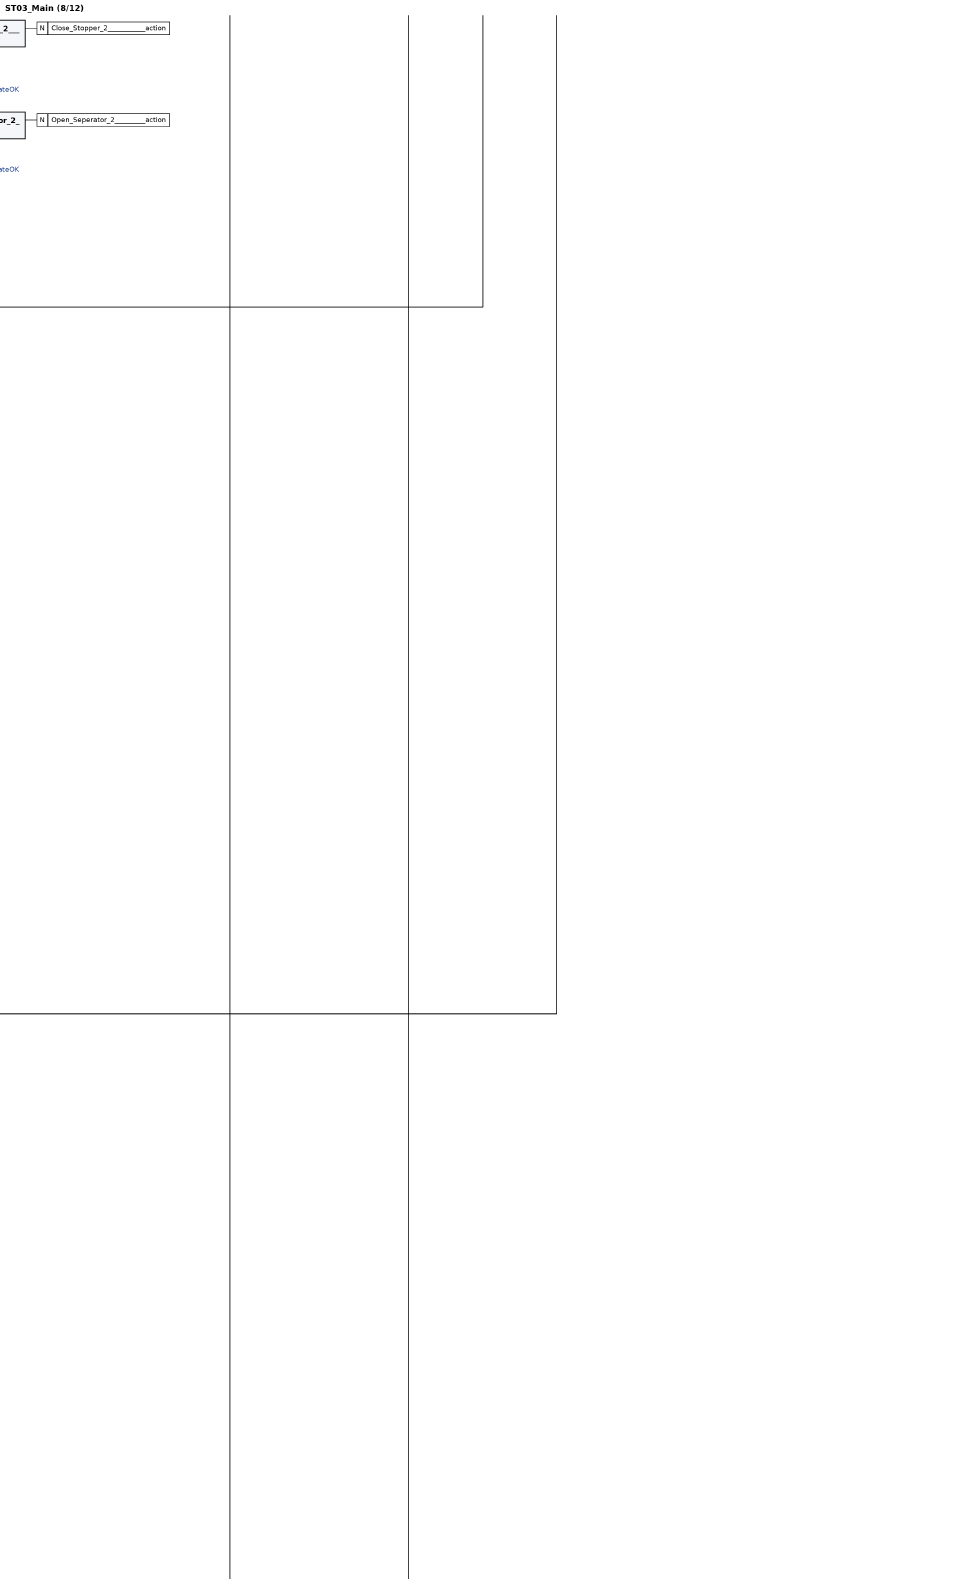
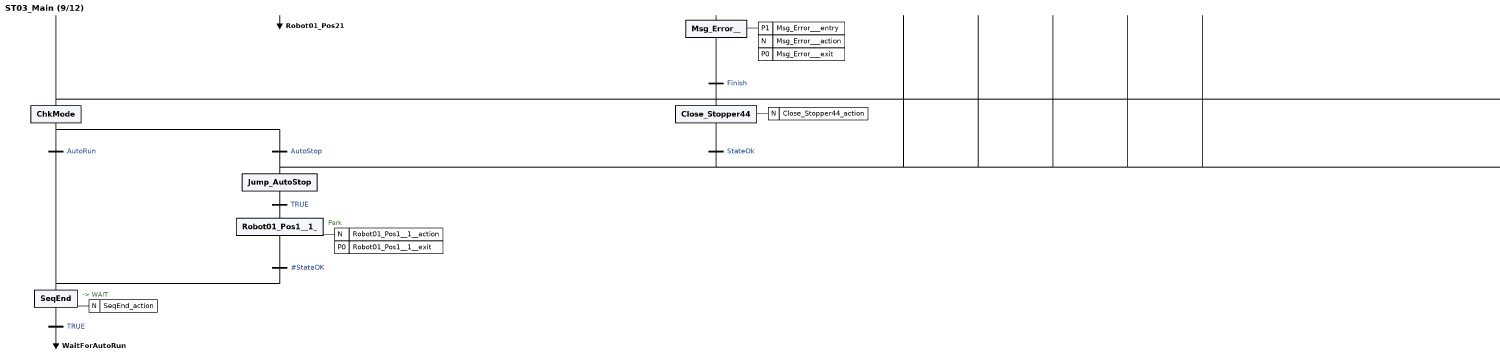
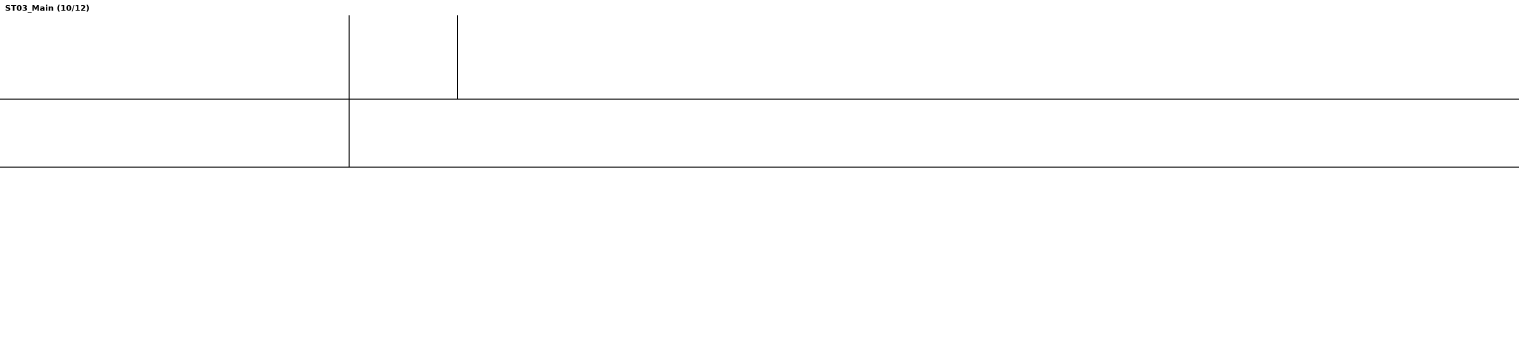
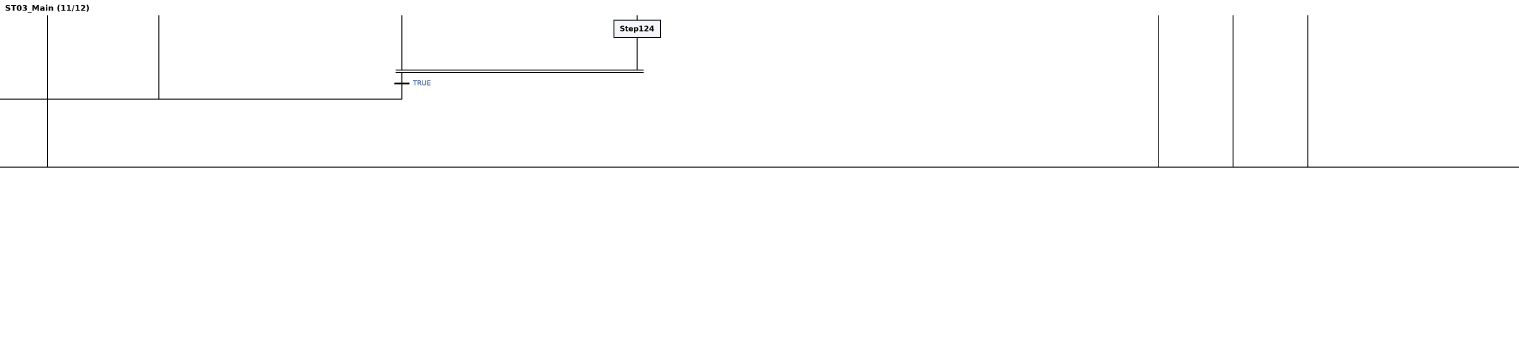
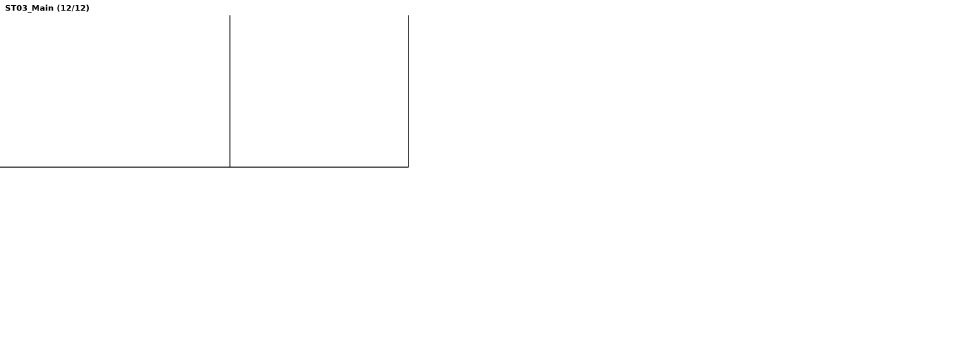
INITIAL_STEP WaitFirstAutRun: (* <-state=AuoRun / ->STATE_RUN *)
	WaitFirstAutRun_action(N);
END_STEP
TRANSITION FROM WaitFirstAutRun TO CheckPartsInRoboGripper := state=2;
END_TRANSITION
STEP CheckPartsInRoboGripper:
END_STEP
TRANSITION FROM CheckPartsInRoboGripper TO ST08_Pallett_ := CheckPartsInRoboGripper;
END_TRANSITION
TRANSITION FROM CheckPartsInRoboGripper TO MsgCheckPartsInRoboGripper := TRUE;
END_TRANSITION
STEP MsgCheckPartsInRoboGripper:
	MsgCheckPartsInRoboGripper_entry(P1);
	MsgCheckPartsInRoboGripper_action(N);
	MsgCheckPartsInRoboGripper_exit(P0);
END_STEP
TRANSITION FROM MsgCheckPartsInRoboGripper TO CheckPartsInRoboGripper := MsgOK;
END_TRANSITION
STEP ST08_Pallett_:
	ST08_Pallett__action(N);
	ST08_Pallett__exit(P0);
END_STEP
TRANSITION FROM ST08_Pallett_ TO Check_Gripper := StateOk;
END_TRANSITION
STEP Check_Gripper:
END_STEP
TRANSITION FROM Check_Gripper TO Robot01_Park := No_Part;
END_TRANSITION
TRANSITION FROM Check_Gripper TO Robot01_PosPal_ := Part_OK_;
END_TRANSITION
TRANSITION FROM Check_Gripper TO Check_RT := Part_New;
END_TRANSITION
TRANSITION FROM Check_Gripper TO Robot01_Park := Part_Cam;
END_TRANSITION
STEP Robot01_PosPal_: (* Put Part / in pal *)
	Robot01_PosPal__entry(P1);
	Robot01_PosPal__action(N);
	Robot01_PosPal__exit(P0);
END_STEP
TRANSITION FROM Robot01_PosPal_ TO ST08_Pallett_2 := StateOK;
END_TRANSITION
STEP ST08_Pallett_2:
	ST08_Pallett_2_action(N);
	ST08_Pallett_2_exit(P0);
END_STEP
TRANSITION FROM ST08_Pallett_2 TO Dummy_Robot := StateOk;
END_TRANSITION
STEP Dummy_Robot:
END_STEP
TRANSITION FROM Dummy_Robot TO Robot01_Pos1___i := TRUE;
END_TRANSITION
STEP Robot01_Pos1___i: (* Park *)
	Robot01_Pos1___i_action(N);
END_STEP
TRANSITION FROM Robot01_Pos1___i TO Check_Type_5 := #StateOK;
END_TRANSITION
STEP Check_RT:
END_STEP
TRANSITION FROM Check_RT TO Jump_IN := RT_Nest_empty;
END_TRANSITION
STEP Robot01_Park: (* Park *)
	Robot01_Park_action(N);
END_STEP
TRANSITION FROM Robot01_Park TO Check_Type_5 := #StateOK;
END_TRANSITION
STEP Check_Type_5:
END_STEP
TRANSITION FROM Check_Type_5 TO WaitForAutoRun := all_other;
END_TRANSITION
TRANSITION FROM Check_Type_5 TO Parts_to_NOK := 93-102polig;
END_TRANSITION
TRANSITION FROM Check_Type_5 TO Open_Stopper := Printer_off;
END_TRANSITION
TRANSITION FROM Check_Type_5 TO WaitForAutoRun := TRUE;
END_TRANSITION
STEP Parts_to_NOK:
	Parts_to_NOK_entry(P1);
	Parts_to_NOK_action(N);
	Parts_to_NOK_exit(P0);
END_STEP
TRANSITION FROM Parts_to_NOK TO TeilNOK := TRUE;
END_TRANSITION
TRANSITION FROM Parts_to_NOK TO WaitForAutoRun := MsgCancel;
END_TRANSITION
STEP TeilNOK:
END_STEP
TRANSITION FROM TeilNOK TO WaitForAutoRun := TRUE;
END_TRANSITION
STEP Open_Stopper:
	Open_Stopper_action(N);
END_STEP
TRANSITION FROM Open_Stopper TO Open_seperator := StateOk;
END_TRANSITION
STEP Open_seperator:
	Open_seperator_action(N);
END_STEP
TRANSITION FROM Open_seperator TO Msg_Error_ := StateOk;
END_TRANSITION
STEP Msg_Error_:
	Msg_Error__entry(P1);
	Msg_Error__action(N);
	Msg_Error__exit(P0);
END_STEP
TRANSITION FROM Msg_Error_ TO Close_Stopper := Finish;
END_TRANSITION
STEP Close_Stopper:
	Close_Stopper_action(N);
END_STEP
TRANSITION FROM Close_Stopper TO Check_Type_5 := StateOk;
END_TRANSITION
STEP WaitForAutoRun: (* -> STATE_RUN *)
	WaitForAutoRun_entry(P1);
	WaitForAutoRun_action(N);
	WaitForAutoRun_exit(P0);
END_STEP
TRANSITION FROM WaitForAutoRun TO Check_Type_ := state = 2;
END_TRANSITION
STEP Check_Type_:
END_STEP
TRANSITION FROM Check_Type_ TO WaitForHandshake := 93_102polig;
END_TRANSITION
TRANSITION FROM Check_Type_ TO WaitCamDone := 268pol;
END_TRANSITION
TRANSITION FROM Check_Type_ TO WaitCamDone_ := 102pol_neu;
END_TRANSITION
TRANSITION FROM Check_Type_ TO Wait_for_Part := all_other_polig;
END_TRANSITION
TRANSITION FROM Check_Type_ TO Check_3621 := T9_74_168_35polig;
END_TRANSITION
STEP WaitCamDone:
END_STEP
TRANSITION FROM WaitCamDone TO TestParts_Activ_ := CamDone;
END_TRANSITION
STEP WaitCamDone_:
END_STEP
TRANSITION FROM WaitCamDone_ TO TestParts_Activ_ := CamDone;
END_TRANSITION
STEP Wait_for_Part: (*  *)
	Wait_for_Part_entry(P1);
	Wait_for_Part_action(N);
	Wait_for_Part_exit(P0);
END_STEP
TRANSITION FROM Wait_for_Part TO WT_POS_1_OR_2_ := Part_Ready_Pick;
END_TRANSITION
TRANSITION FROM Wait_for_Part TO Jump_AutoStop := AutoStop;
END_TRANSITION
STEP WT_POS_1_OR_2_:
END_STEP
TRANSITION FROM WT_POS_1_OR_2_ TO Robot01_Pos31_5 := POS_1;
END_TRANSITION
TRANSITION FROM WT_POS_1_OR_2_ TO Robot01_Pos35__ := POS_2;
END_TRANSITION
STEP Robot01_Pos35__: (* Pick Part / from Belt *)
	Robot01_Pos35___action(N);
	Robot01_Pos35___exit(P0);
END_STEP
TRANSITION FROM Robot01_Pos35__ TO TestParts_Activ_ := #StateOK;
END_TRANSITION
STEP Robot01_Pos31_5: (* Pick Part / from Belt *)
	Robot01_Pos31_5_action(N);
	Robot01_Pos31_5_exit(P0);
END_STEP
TRANSITION FROM Robot01_Pos31_5 TO TestParts_Activ_ := #StateOK;
END_TRANSITION
STEP TestParts_Activ_:
	TestParts_Activ__action(N);
END_STEP
TRANSITION FROM TestParts_Activ_ TO Robot01_TestPos_ := Yes;
END_TRANSITION
TRANSITION FROM TestParts_Activ_ TO ST08_Pallett_53 := i.O.;
END_TRANSITION
TRANSITION FROM TestParts_Activ_ TO Robot01_Pos51 := n.i.O;
END_TRANSITION
STEP ST08_Pallett_53:
	ST08_Pallett_53_entry(P1);
	ST08_Pallett_53_action(N);
	ST08_Pallett_53_exit(P0);
END_STEP
TRANSITION FROM ST08_Pallett_53 TO Pal_Ready_5 := StateOk;
END_TRANSITION
TRANSITION FROM ST08_Pallett_53 TO Robot01_POS_PARK_ := TRUE;
END_TRANSITION
STEP Robot01_POS_PARK_: (* Warte über / POS_PARK *)
	Robot01_POS_PARK__action(N);
END_STEP
TRANSITION FROM Robot01_POS_PARK_ TO Pal_Ready_5 := StateOk;
END_TRANSITION
STEP Pal_Ready_5:
END_STEP
TRANSITION FROM Pal_Ready_5 TO Robot01_PosPal_5 := Pal_OK;
END_TRANSITION
TRANSITION FROM Pal_Ready_5 TO Stecker91Pol := TRUE;
END_TRANSITION
STEP Stecker91Pol:
END_STEP
TRANSITION FROM Stecker91Pol TO Release_Nest_2 := allOther;
END_TRANSITION
TRANSITION FROM Stecker91Pol TO Robi_PallWait := TRUE;
END_TRANSITION
STEP Robi_PallWait:
	Robi_PallWait_action(N);
END_STEP
TRANSITION FROM Robi_PallWait TO Release_Nest_2 := StateOk;
END_TRANSITION
STEP Release_Nest_2:
	Release_Nest_2_action(N);
END_STEP
TRANSITION FROM Release_Nest_2 TO ST08_Pallett_5 := OK;
END_TRANSITION
STEP ST08_Pallett_5:
	ST08_Pallett_5_entry(P1);
	ST08_Pallett_5_action(N);
	ST08_Pallett_5_exit(P0);
END_STEP
TRANSITION FROM ST08_Pallett_5 TO Pal_Ready_51 := StateOk;
END_TRANSITION
STEP Pal_Ready_51:
END_STEP
TRANSITION FROM Pal_Ready_51 TO Robot01_PosPal_5 := Pal_OK;
END_TRANSITION
STEP Robot01_PosPal_5: (* Put Part / in pal *)
	Robot01_PosPal_5_entry(P1);
	Robot01_PosPal_5_action(N);
	Robot01_PosPal_5_exit(P0);
END_STEP
TRANSITION FROM Robot01_PosPal_5 TO Reset_Test2 := StateOK;
END_TRANSITION
STEP Reset_Test2:
	Reset_Test2_action(N);
END_STEP
TRANSITION FROM Reset_Test2 TO Release_Nest_21 := TRUE;
END_TRANSITION
STEP Release_Nest_21:
	Release_Nest_21_action(N);
END_STEP
TRANSITION FROM Release_Nest_21 TO ST08_Pallett_51 := OK;
END_TRANSITION
STEP ST08_Pallett_51:
	ST08_Pallett_51_action(N);
END_STEP
TRANSITION FROM ST08_Pallett_51 TO Robot01_POS_PARK_12 := StateRun;
END_TRANSITION
STEP Robot01_Pos51: (* go to Nio *)
	Robot01_Pos51_action(N);
END_STEP
TRANSITION FROM Robot01_Pos51 TO Delay___ := #StateOK;
END_TRANSITION
STEP Delay___: (* min time t#1000ms; t#1000ms *)
END_STEP
TRANSITION FROM Delay___ TO Robot01_POS_PARK_12 := TRUE;
END_TRANSITION
STEP Robot01_TestPos_:
	Robot01_TestPos__entry(P1);
	Robot01_TestPos__action(N);
	Robot01_TestPos__exit(P0);
END_STEP
TRANSITION FROM Robot01_TestPos_ TO Reset_Test_ := StateOK;
END_TRANSITION
STEP Reset_Test_:
	Reset_Test__action(N);
END_STEP
TRANSITION FROM Reset_Test_ TO Robot01_POS_PARK_12 := empty;
END_TRANSITION
STEP Robot01_POS_PARK_12: (* Warte über / POS_PARK *)
	Robot01_POS_PARK_12_action(N);
END_STEP
TRANSITION FROM Robot01_POS_PARK_12 TO ChkMode := #StateOK;
END_TRANSITION
STEP Check_3621:
END_STEP
TRANSITION FROM Check_3621 TO Checxk_Abholpos := all_other;
END_TRANSITION
TRANSITION FROM Check_3621 TO Chech_Abolpos := SGM_3621;
END_TRANSITION
STEP Chech_Abolpos:
END_STEP
TRANSITION FROM Chech_Abolpos TO Close_Stopper___________ := leer;
END_TRANSITION
TRANSITION FROM Chech_Abolpos TO WT_POS1_OR_2 := true;
END_TRANSITION
STEP Close_Stopper___________:
	Close_Stopper____________action(N);
END_STEP
TRANSITION FROM Close_Stopper___________ TO Open_Seperator_________ := StateOK;
END_TRANSITION
STEP Open_Seperator_________:
	Open_Seperator__________action(N);
END_STEP
TRANSITION FROM Open_Seperator_________ TO Wait__for_Part____ := StateOK;
END_TRANSITION
STEP Wait__for_Part____: (*  *)
	Wait__for_Part_____entry(P1);
	Wait__for_Part_____action(N);
	Wait__for_Part_____exit(P0);
END_STEP
TRANSITION FROM Wait__for_Part____ TO Close__seperator_ := Part_Ready_Print;
END_TRANSITION
TRANSITION FROM Wait__for_Part____ TO Jump_AutoStop := AutoStop;
END_TRANSITION
STEP Close__seperator_:
	Close__seperator__action(N);
END_STEP
TRANSITION FROM Close__seperator_ TO Open__Stopper__ := StateOk;
END_TRANSITION
STEP Open__Stopper__:
	Open__Stopper___action(N);
END_STEP
TRANSITION FROM Open__Stopper__ TO Wait_for__Part__ := StateOk;
END_TRANSITION
STEP Wait_for__Part__:
	Wait_for__Part___entry(P1);
	Wait_for__Part___action(N);
	Wait_for__Part___exit(P0);
END_STEP
TRANSITION FROM Wait_for__Part__ TO Close_Stopper_2__________ := Part_Ready_Roboter;
END_TRANSITION
TRANSITION FROM Wait_for__Part__ TO Jump_AutoStop := AutoStop;
END_TRANSITION
STEP Close_Stopper_2__________:
	Close_Stopper_2___________action(N);
END_STEP
TRANSITION FROM Close_Stopper_2__________ TO Open_Seperator_2________ := StateOK;
END_TRANSITION
STEP Open_Seperator_2________:
	Open_Seperator_2_________action(N);
END_STEP
TRANSITION FROM Open_Seperator_2________ TO Step120 := StateOK;
END_TRANSITION
STEP Checxk_Abholpos:
END_STEP
TRANSITION FROM Checxk_Abholpos TO Close_Stopper_ := Abholpos_leer;
END_TRANSITION
TRANSITION FROM Checxk_Abholpos TO WT_POS1_OR_2 := TRUE;
END_TRANSITION
STEP Close_Stopper_:
	Close_Stopper__action(N);
END_STEP
TRANSITION FROM Close_Stopper_ TO Open_seperator_ := StateOk;
END_TRANSITION
STEP Open_seperator_:
	Open_seperator__action(N);
END_STEP
TRANSITION FROM Open_seperator_ TO Wait_for_Part_ := StateOk;
END_TRANSITION
STEP Wait_for_Part_: (*  *)
	Wait_for_Part__entry(P1);
	Wait_for_Part__action(N);
	Wait_for_Part__exit(P0);
END_STEP
TRANSITION FROM Wait_for_Part_ TO Move_Dist := Part_Ready_Print;
END_TRANSITION
TRANSITION FROM Wait_for_Part_ TO Jump_AutoStop := AutoStop;
END_TRANSITION
STEP Move_Dist:
	Move_Dist_entry(P1);
END_STEP
TRANSITION FROM Move_Dist TO Close_seperator_ := Wait_Pos;
END_TRANSITION
STEP Close_seperator_:
	Close_seperator__action(N);
END_STEP
TRANSITION FROM Close_seperator_ TO Open_Stopper__ := StateOk;
END_TRANSITION
STEP Open_Stopper__:
	Open_Stopper___action(N);
END_STEP
TRANSITION FROM Open_Stopper__ TO Wait_for_Part__ := StateOk;
END_TRANSITION
STEP Wait_for_Part__:
	Wait_for_Part___entry(P1);
	Wait_for_Part___action(N);
	Wait_for_Part___exit(P0);
END_STEP
TRANSITION FROM Wait_for_Part__ TO Close_Stopper______ := Part_Ready_Roboter;
END_TRANSITION
TRANSITION FROM Wait_for_Part__ TO Jump_AutoStop := AutoStop;
END_TRANSITION
STEP Close_Stopper______:
	Close_Stopper_______action(N);
END_STEP
TRANSITION FROM Close_Stopper______ TO Open_seperator______ := StateOk;
END_TRANSITION
STEP Open_seperator______:
	Open_seperator_______action(N);
END_STEP
TRANSITION FROM Open_seperator______ TO Step120 := StateOk;
END_TRANSITION
STEP Step120:
END_STEP
TRANSITION FROM Step120 TO WT_POS1_OR_2 := TRUE;
END_TRANSITION
STEP WT_POS1_OR_2:
END_STEP
TRANSITION FROM WT_POS1_OR_2 TO Stopp_Band_91pol := not_35pol_or_links;
END_TRANSITION
TRANSITION FROM WT_POS1_OR_2 TO Robot01_Pos35 := 35pol_rechts;
END_TRANSITION
STEP Robot01_Pos35: (* Pick Part / from Belt right *)
	Robot01_Pos35_action(N);
	Robot01_Pos35_exit(P0);
END_STEP
TRANSITION FROM Robot01_Pos35 TO delay2 := #StateOK;
END_TRANSITION
STEP Stopp_Band_91pol:
	Stopp_Band_91pol_action(N);
END_STEP
TRANSITION FROM Stopp_Band_91pol TO Robot01_Pos31_65 := TRUE;
END_TRANSITION
STEP Robot01_Pos31_65: (* Pick Part / from Belt left *)
	Robot01_Pos31_65_action(N);
	Robot01_Pos31_65_exit(P0);
END_STEP
TRANSITION FROM Robot01_Pos31_65 TO Band_starten := #StateOK;
END_TRANSITION
STEP Band_starten:
	Band_starten_action(N);
END_STEP
TRANSITION FROM Band_starten TO delay2 := TRUE;
END_TRANSITION
STEP delay2: (* min time t#50ms; t#50ms *)
END_STEP
TRANSITION FROM delay2 TO Robot01__POS_PARK := TRUE;
END_TRANSITION
STEP Robot01__POS_PARK: (* Warte über / POS_PARK *)
	Robot01__POS_PARK_action(N);
END_STEP
TRANSITION FROM Robot01__POS_PARK TO TestParts_Activ___ := #StateOK;
END_TRANSITION
STEP TestParts_Activ___:
END_STEP
TRANSITION FROM TestParts_Activ___ TO Robot01_TestPos__ := Yes;
END_TRANSITION
TRANSITION FROM TestParts_Activ___ TO ST08_Pallett_6 := No;
END_TRANSITION
STEP ST08_Pallett_6:
	ST08_Pallett_6_entry(P1);
	ST08_Pallett_6_action(N);
	ST08_Pallett_6_exit(P0);
END_STEP
TRANSITION FROM ST08_Pallett_6 TO Pal_Ready_6 := StateOk;
END_TRANSITION
TRANSITION FROM ST08_Pallett_6 TO Pal_Ready_6 := StateWait;
END_TRANSITION
STEP Pal_Ready_6:
END_STEP
TRANSITION FROM Pal_Ready_6 TO (Robot01_PosPal_65, Iso_an_Vereinzler) := Pal_OK;
END_TRANSITION
TRANSITION FROM Pal_Ready_6 TO Jump_AutoStop := AutoStop;
END_TRANSITION
STEP Robot01_PosPal_65: (* Put Part / in pal *)
	Robot01_PosPal_65_entry(P1);
	Robot01_PosPal_65_action(N);
	Robot01_PosPal_65_exit(P0);
END_STEP
TRANSITION FROM Robot01_PosPal_65 TO Reset_Test3 := StateOK;
END_TRANSITION
STEP Reset_Test3:
	Reset_Test3_action(N);
END_STEP
TRANSITION FROM Reset_Test3 TO ST08_Pallett_8 := TRUE;
END_TRANSITION
STEP ST08_Pallett_8:
	ST08_Pallett_8_action(N);
END_STEP
TRANSITION FROM ST08_Pallett_8 TO Robot01_POS_PARK_3_ := StateRun;
END_TRANSITION
STEP Robot01_POS_PARK_3_: (* Warte über / POS_PARK *)
	Robot01_POS_PARK_3__action(N);
END_STEP
TRANSITION FROM Robot01_POS_PARK_3_ TO Step123 := #StateOK;
END_TRANSITION
STEP Step123:
END_STEP
STEP Iso_an_Vereinzler:
END_STEP
TRANSITION FROM Iso_an_Vereinzler TO ActualArea := Iso_an_Vereinzler;
END_TRANSITION
TRANSITION FROM Iso_an_Vereinzler TO Step124 := TRUE;
END_TRANSITION
STEP ActualArea:
END_STEP
TRANSITION FROM ActualArea TO _Check_3621_1 := Trans151;
END_TRANSITION
STEP _Check_3621_1:
END_STEP
TRANSITION FROM _Check_3621_1 TO Close_seperator__ := all_other;
END_TRANSITION
TRANSITION FROM _Check_3621_1 TO Close__seperator_2 := SGM_3621;
END_TRANSITION
STEP Close__seperator_2:
	Close__seperator_2_action(N);
END_STEP
TRANSITION FROM Close__seperator_2 TO Open__Stopper_2_ := StateOk;
END_TRANSITION
STEP Open__Stopper_2_:
	Open__Stopper_2__action(N);
END_STEP
TRANSITION FROM Open__Stopper_2_ TO Wait_for_Part___ := StateOk;
END_TRANSITION
STEP Wait_for_Part___:
	Wait_for_Part____entry(P1);
	Wait_for_Part____action(N);
	Wait_for_Part____exit(P0);
END_STEP
TRANSITION FROM Wait_for_Part___ TO Close_Stopper_1__________ := Part_Ready_Roboter;
END_TRANSITION
STEP Close_Stopper_1__________:
	Close_Stopper_1___________action(N);
END_STEP
TRANSITION FROM Close_Stopper_1__________ TO Open_Seperator_1________ := StateOK;
END_TRANSITION
STEP Open_Seperator_1________:
	Open_Seperator_1_________action(N);
END_STEP
TRANSITION FROM Open_Seperator_1________ TO Step124 := StateOK;
END_TRANSITION
STEP Close_seperator__:
	Close_seperator___action(N);
END_STEP
TRANSITION FROM Close_seperator__ TO Open_Stopper___ := StateOk;
END_TRANSITION
STEP Open_Stopper___:
	Open_Stopper____action(N);
END_STEP
TRANSITION FROM Open_Stopper___ TO Wait_for_Part_1__ := StateOk;
END_TRANSITION
STEP Wait_for_Part_1__:
	Wait_for_Part_1___entry(P1);
	Wait_for_Part_1___action(N);
	Wait_for_Part_1___exit(P0);
END_STEP
TRANSITION FROM Wait_for_Part_1__ TO Close__Stopper______ := Part_Ready_Roboter;
END_TRANSITION
STEP Close__Stopper______:
	Close__Stopper_______action(N);
END_STEP
TRANSITION FROM Close__Stopper______ TO Open_seperator___ := StateOk;
END_TRANSITION
STEP Open_seperator___:
	Open_seperator____action(N);
END_STEP
TRANSITION FROM Open_seperator___ TO Step124 := StateOk;
END_TRANSITION
STEP Step124:
END_STEP
TRANSITION FROM (Step123, Step124) TO ChkMode := TRUE;
END_TRANSITION
STEP Robot01_TestPos__:
	Robot01_TestPos___entry(P1);
	Robot01_TestPos___action(N);
	Robot01_TestPos___exit(P0);
END_STEP
TRANSITION FROM Robot01_TestPos__ TO Reset_Test__ := StateOK;
END_TRANSITION
STEP Reset_Test__:
	Reset_Test___action(N);
END_STEP
TRANSITION FROM Reset_Test__ TO Robot01_POS_PARK_3 := TRUE;
END_TRANSITION
STEP Robot01_POS_PARK_3: (* Warte über / POS_PARK *)
	Robot01_POS_PARK_3_action(N);
END_STEP
TRANSITION FROM Robot01_POS_PARK_3 TO ChkMode := #StateOK;
END_TRANSITION
STEP WaitForHandshake: (*  *)
END_STEP
TRANSITION FROM WaitForHandshake TO Robot01_Pos21 := Part_Ready_Print;
END_TRANSITION
TRANSITION FROM WaitForHandshake TO Check_ST02_Main_Print := RT_Nest_empty;
END_TRANSITION
TRANSITION FROM WaitForHandshake TO Jump_AutoStop := AutoStop;
END_TRANSITION
STEP Check_ST02_Main_Print:
END_STEP
TRANSITION FROM Check_ST02_Main_Print TO Part_Ready_Belt := Wait_;
END_TRANSITION
TRANSITION FROM Check_ST02_Main_Print TO ST02_Main_Print := TRUE;
END_TRANSITION
STEP ST02_Main_Print: (* SFC *)
	ST02_Main_Print_exit(P0);
END_STEP
TRANSITION FROM ST02_Main_Print TO Part_Ready_Belt := StateOk;
END_TRANSITION
STEP Robot01_Pos21: (* Pick Part / from Printer *)
	Robot01_Pos21_action(N);
	Robot01_Pos21_exit(P0);
END_STEP
TRANSITION FROM Robot01_Pos21 TO set_PartState := #StateOK;
END_TRANSITION
STEP set_PartState:
	set_PartState_exit(P0);
END_STEP
TRANSITION FROM set_PartState TO TestParts_Activ := CounterCheck;
END_TRANSITION
TRANSITION FROM set_PartState TO Robo01_PosNOK := TRUE;
END_TRANSITION
STEP Robo01_PosNOK:
	Robo01_PosNOK_action(N);
	Robo01_PosNOK_exit(P0);
END_STEP
TRANSITION FROM Robo01_PosNOK TO Check_SFC_Print := #StateOK;
END_TRANSITION
STEP TestParts_Activ:
END_STEP
TRANSITION FROM TestParts_Activ TO RampFree := Yes;
END_TRANSITION
TRANSITION FROM TestParts_Activ TO ST08_Pallett_33 := No;
END_TRANSITION
STEP ST08_Pallett_33:
	ST08_Pallett_33_entry(P1);
	ST08_Pallett_33_action(N);
	ST08_Pallett_33_exit(P0);
END_STEP
TRANSITION FROM ST08_Pallett_33 TO Pal_Ready := StateOk;
END_TRANSITION
TRANSITION FROM ST08_Pallett_33 TO Pal_Ready := StateWait;
END_TRANSITION
STEP Pal_Ready:
END_STEP
TRANSITION FROM Pal_Ready TO Robot01_PosPal := Pal_OK;
END_TRANSITION
TRANSITION FROM Pal_Ready TO Robot01_POS_PARK := TRUE;
END_TRANSITION
STEP Robot01_POS_PARK: (* Warte über / POS_PARK *)
	Robot01_POS_PARK_action(N);
END_STEP
TRANSITION FROM Robot01_POS_PARK TO ST08_Pallett_3 := #StateOK;
END_TRANSITION
STEP ST08_Pallett_3:
	ST08_Pallett_3_entry(P1);
	ST08_Pallett_3_action(N);
	ST08_Pallett_3_exit(P0);
END_STEP
TRANSITION FROM ST08_Pallett_3 TO Pal_Ready_ := StateOk;
END_TRANSITION
STEP Pal_Ready_:
END_STEP
TRANSITION FROM Pal_Ready_ TO Robot01_PosPal := Pal_OK;
END_TRANSITION
STEP Robot01_PosPal:
	Robot01_PosPal_entry(P1);
	Robot01_PosPal_action(N);
	Robot01_PosPal_exit(P0);
END_STEP
TRANSITION FROM Robot01_PosPal TO Reset_Test1 := StateOK;
END_TRANSITION
STEP Reset_Test1:
	Reset_Test1_action(N);
END_STEP
TRANSITION FROM Reset_Test1 TO ST08_Pallett := TRUE;
END_TRANSITION
STEP ST08_Pallett:
	ST08_Pallett_action(N);
END_STEP
TRANSITION FROM ST08_Pallett TO Robot01_POS32_ := StateRun;
END_TRANSITION
STEP RampFree:
END_STEP
TRANSITION FROM RampFree TO Robot01_TestPos := Yes;
END_TRANSITION
TRANSITION FROM RampFree TO RemoveTestParts := TRUE;
END_TRANSITION
STEP RemoveTestParts:
	RemoveTestParts_entry(P1);
	RemoveTestParts_action(N);
	RemoveTestParts_exit(P0);
END_STEP
TRANSITION FROM RemoveTestParts TO Robot01_TestPos := MsgOk;
END_TRANSITION
STEP Robot01_TestPos: (* Ablage Test / Part *)
	Robot01_TestPos_entry(P1);
	Robot01_TestPos_action(N);
	Robot01_TestPos_exit(P0);
END_STEP
TRANSITION FROM Robot01_TestPos TO Step137 := StateOK;
END_TRANSITION
STEP Step137:
END_STEP
TRANSITION FROM Step137 TO Reset_Test := all_other___;
END_TRANSITION
TRANSITION FROM Step137 TO Step140 := Last_Dummy;
END_TRANSITION
STEP Step140:
	Step140_action(N);
END_STEP
TRANSITION FROM Step140 TO Robot01_Pos21___ := Part_Ready___;
END_TRANSITION
STEP Robot01_Pos21___: (* Pick Part / from Printer *)
	Robot01_Pos21____action(N);
	Robot01_Pos21____exit(P0);
END_STEP
TRANSITION FROM Robot01_Pos21___ TO Robot01_Pos21 := #StateOK;
END_TRANSITION
STEP Reset_Test:
	Reset_Test_action(N);
END_STEP
TRANSITION FROM Reset_Test TO Robot01_POS32_ := TRUE;
END_TRANSITION
STEP Robot01_POS32_: (* Warte über / Band *)
	Robot01_POS32__action(N);
END_STEP
TRANSITION FROM Robot01_POS32_ TO Check_SFC_Print := #StateOK;
END_TRANSITION
TRANSITION FROM Robot01_POS32_ TO Jump_AutoStop := AutoStop;
END_TRANSITION
STEP Check_SFC_Print:
END_STEP
TRANSITION FROM Check_SFC_Print TO Check_Mode_Run := TRUE;
END_TRANSITION
STEP Check_Mode_Run:
END_STEP
TRANSITION FROM Check_Mode_Run TO Part_Ready_Belt := Auto_run;
END_TRANSITION
TRANSITION FROM Check_Mode_Run TO Jump_AutoStop := AutoStop;
END_TRANSITION
STEP Part_Ready_Belt:
END_STEP
TRANSITION FROM Part_Ready_Belt TO Robot01_Pos31 := PartReady;
END_TRANSITION
STEP Robot01_Pos31: (* Pick Part / from Belt *)
	Robot01_Pos31_action(N);
	Robot01_Pos31_exit(P0);
END_STEP
TRANSITION FROM Robot01_Pos31 TO Dummy_Robot___ := #StateOK;
END_TRANSITION
STEP Dummy_Robot___: (* min time T#300ms; T#300ms *)
END_STEP
TRANSITION FROM Dummy_Robot___ TO Robot01_POS22 := TRUE;
END_TRANSITION
STEP Robot01_POS22: (* Warte über / RT *)
	Robot01_POS22_action(N);
END_STEP
TRANSITION FROM Robot01_POS22 TO Put_in_RT_2 := #StateOK;
END_TRANSITION
STEP Put_in_RT_2:
END_STEP
TRANSITION FROM Put_in_RT_2 TO Handshake := TRUE;
END_TRANSITION
STEP Handshake:
	Handshake_entry(P1);
	Handshake_exit(P0);
END_STEP
TRANSITION FROM Handshake TO Jump_IN := OK;
END_TRANSITION
TRANSITION FROM Handshake TO Jump_AutoStop := AutoStop;
END_TRANSITION
STEP Jump_IN:
END_STEP
TRANSITION FROM Jump_IN TO Robot01_Pos21_ := Part_Ready_Print;
END_TRANSITION
TRANSITION FROM Jump_IN TO Jump_AutoStop := AutoStop;
END_TRANSITION
STEP Robot01_Pos21_: (* Put Part / in Printer *)
	Robot01_Pos21__action(N);
	Robot01_Pos21__exit(P0);
END_STEP
TRANSITION FROM Robot01_Pos21_ TO set_PartState_ := #StateOK;
END_TRANSITION
STEP set_PartState_:
	set_PartState__exit(P0);
END_STEP
TRANSITION FROM set_PartState_ TO Robot01_POS23_ := TRUE;
END_TRANSITION
STEP Robot01_POS23_: (* Warte vor / RT *)
	Robot01_POS23__action(N);
END_STEP
TRANSITION FROM Robot01_POS23_ TO Step136 := #StateOK;
END_TRANSITION
STEP Step136:
END_STEP
TRANSITION FROM Step136 TO ST02_Main_Print_ := ST02Wait;
END_TRANSITION
STEP ST02_Main_Print_: (* SFC *)
	ST02_Main_Print__action(N);
	ST02_Main_Print__exit(P0);
END_STEP
TRANSITION FROM ST02_Main_Print_ TO Wait_Printer_finish_ := turn_done;
END_TRANSITION
STEP Wait_Printer_finish_: (* warte auf / Drucker fertig *)
	Wait_Printer_finish__entry(P1);
	Wait_Printer_finish__action(N);
	Wait_Printer_finish__exit(P0);
END_STEP
TRANSITION FROM Wait_Printer_finish_ TO Fertig := IO;
END_TRANSITION
TRANSITION FROM Wait_Printer_finish_ TO NIO := NIO;
END_TRANSITION
TRANSITION FROM Wait_Printer_finish_ TO Part_Ready_Belt := emty;
END_TRANSITION
TRANSITION FROM Wait_Printer_finish_ TO Open_Stopper3 := Time_out;
END_TRANSITION
TRANSITION FROM Wait_Printer_finish_ TO Jump_AutoStop := AutoStop;
END_TRANSITION
STEP NIO:
END_STEP
TRANSITION FROM NIO TO Robot01_Pos21 := TRUE;
END_TRANSITION
STEP Open_Stopper3:
	Open_Stopper3_action(N);
END_STEP
TRANSITION FROM Open_Stopper3 TO Msg_Error__ := StateOk;
END_TRANSITION
STEP Msg_Error__:
	Msg_Error___entry(P1);
	Msg_Error___action(N);
	Msg_Error___exit(P0);
END_STEP
TRANSITION FROM Msg_Error__ TO Close_Stopper44 := Finish;
END_TRANSITION
STEP Close_Stopper44:
	Close_Stopper44_action(N);
END_STEP
TRANSITION FROM Close_Stopper44 TO Jump_AutoStop := StateOk;
END_TRANSITION
STEP Fertig:
	Fertig_entry(P1);
END_STEP
TRANSITION FROM Fertig TO ChkMode := TRUE;
END_TRANSITION
STEP ChkMode:
END_STEP
TRANSITION FROM ChkMode TO SeqEnd := AutoRun;
END_TRANSITION
TRANSITION FROM ChkMode TO Jump_AutoStop := AutoStop;
END_TRANSITION
STEP Jump_AutoStop:
END_STEP
TRANSITION FROM Jump_AutoStop TO Robot01_Pos1__1_ := TRUE;
END_TRANSITION
STEP Robot01_Pos1__1_: (* Park *)
	Robot01_Pos1__1__action(N);
	Robot01_Pos1__1__exit(P0);
END_STEP
TRANSITION FROM Robot01_Pos1__1_ TO SeqEnd := #StateOK;
END_TRANSITION
STEP SeqEnd: (* -> WAIT *)
	SeqEnd_action(N);
END_STEP
TRANSITION FROM SeqEnd TO WaitForAutoRun := TRUE;
END_TRANSITION

ACTION WaitFirstAutRun_action:
IF 	ModeSelect.Mode=MODE_AUTO_RUN OR
	ModeSelect.Mode=MODE_STEP_RUN OR
	(SpecialMode06.State=State_Run AND
	(gTypeCode=312 OR			(*93pol*)
	gTypeCode=499)) 			(*102pol*)
THEN
	State:=STATE_RUN;
ELSE
	State:=STATE_WAIT;
	MsgOK:=FALSE;
	MsgCancel:=FALSE;
	SFCRun:=FALSE;
END_IF

Nest10Locked:=FALSE;
Nest10Done:=FALSE;
Side_1:=FALSE;
Side_2:=FALSE;
PutIdx:=0;
Nest_Empty:=FALSE;
ST03_Autostop.Start:=FALSE;
CTR:=0;
CTR2:=0;
END_ACTION

ACTION MsgCheckPartsInRoboGripper_entry:
MessageHandler.ClearMessageLines(sVisu:=Visu.Message);
MsgOk := FALSE;
END_ACTION

ACTION MsgCheckPartsInRoboGripper_action:
MessageHandler.Msg.ID:='PM121';
MessageHandler.Msg.Name:='Anzahl Teile im Greifer darf nicht 0 sein';
MessageHandler.Msg.Text:= 'Anzahl Teile im Greifer darf nicht 0 sein ';
MessageHandler.Msg.Color:=Color.red;
MessageHandler.Msg.Station:=1;

MessageHandler(
	Prio:=2, 								(*1=highest, .. , 4=lowest*)
	Btn1Addr:=ADR(MsgOk),		(*Address of Button1 , if Zero then Button is unvisible*)
	Btn2Addr:=0,						(*Address of Button2 , if Zero then Button is unvisible*)
	sVisu:=Visu.Message);
END_ACTION

ACTION MsgCheckPartsInRoboGripper_exit:
MsgOk := FALSE;
END_ACTION

ACTION ST08_Pallett__action:
IF 	ST08_Process.State=STATE_WAIT THEN
	ST08_Process.Start:=TRUE;
END_IF
END_ACTION

ACTION ST08_Pallett__exit:
ST08_Process.Start:=FALSE;
END_ACTION

ACTION Robot01_PosPal__entry:
IF 	PosIdx<TD.PartsInRoboGripper THEN
	PosIdx:=TD.PartsInRoboGripper;
END_IF
END_ACTION

ACTION Robot01_PosPal__action:
Robot01.PosNo:=POS_FEED_PAL_WAIT + (PosIdx/TD.PartsInRoboGripper);
Robot01.PosOffset:=gRobotOffset;
Robot01.Override:=MP.ST00.Override;
Robot01.SetToolOn:=TRUE;
Robot01.SetToolOff:=FALSE;
Robot01.ExecuteMove:=TRUE;
END_ACTION

ACTION Robot01_PosPal__exit:
gRob01GripState:=PART_NO;
PosIdx:=PosIdx+TD.PartsInRoboGripper;
gPartsInserted:=gPartsInserted+TD.PartsInRoboGripper;
gPartsTest:=gPartsTest+TD.PartsInRoboGripper;
END_ACTION

ACTION ST08_Pallett_2_action:
IF 	ST08_Process.State=STATE_WAIT THEN
	ST08_Process.Start:=TRUE;
END_IF
END_ACTION

ACTION ST08_Pallett_2_exit:
ST08_Process.Start:=FALSE;
END_ACTION

ACTION Robot01_Pos1___i_action:
Robot01.PosNo:=POS_PARK;
Robot01.PosOffset:=gRobotOffset;
Robot01.Override:=MP.ST00.Override;
(*Robot01.SetToolOn:=TRUE;
Robot01.SetToolOff:=FALSE;*)
Robot01.ExecuteMove:=TRUE;
END_ACTION

ACTION Robot01_Park_action:
Robot01.PosNo:=POS_PARK;
Robot01.PosOffset:=gRobotOffset;
Robot01.Override:=MP.ST00.Override;
Robot01.SetToolOn:=TRUE;
Robot01.SetToolOff:=FALSE;
Robot01.ExecuteMove:=TRUE;
END_ACTION

ACTION Parts_to_NOK_entry:
MessageHandler.ClearMessageLines(sVisu:=Visu.Message);
END_ACTION

ACTION Parts_to_NOK_action:
MessageHandler.Msg.ID:='PM114';
MessageHandler.Msg.Name:='Start Stecker 93polig';
MessageHandler.Msg.Text:='Solllen die ersten Teile auf NOK pos gelegt werden -> mit OK$R';
MessageHandler.Msg.Text:=CONCAT(MessageHandler.Msg.Text,'-> Abbrechen, sofort in Palettierer');
MessageHandler.Msg.Color:=Color.yellow;
MessageHandler.Msg.Station:=1;


MessageHandler(
	Prio:=2, 									(*1=highest, .. , 4=lowest*)
	Btn1Addr:=ADR(MsgOk),			(*Address of Button1 , if Zero then Button is unvisible*)
	Btn2Addr:=ADR(MsgCancel),	(*Address of Button2 , if Zero then Button is unvisible*)
	sVisu:=Visu.Message);


MessageHandler.MessageLine[1].Visible:=TRUE;
MessageHandler.MessageLine[1].Editable:=TRUE;
MessageHandler.MessageLine[1].Text:='Anzahl Teile auf NOK';
MessageHandler.MessageLine[1].MsgTypeEnum:=MsgDataTypeDint;
END_ACTION

ACTION Parts_to_NOK_exit:
MsgOk:=FALSE;
MsgCancel:=FALSE;
AnzahlTeile:=MessageHandler.MessageLine[1].MsgInt;

(*erstes Teil soll immer in nok Box*)
IF AnzahlTeile < 3 THEN
	AnzahlTeile := 3;
END_IF
END_ACTION

ACTION Open_Stopper_action:
ST00_74_Y2_4.MoveWork:=TRUE;
END_ACTION

ACTION Open_seperator_action:
ST00_74_Y2_5.MoveInit:=TRUE;
END_ACTION

ACTION Msg_Error__entry:
MessageHandler.ClearMessageLines(sVisu:=Visu.Message);
END_ACTION

ACTION Msg_Error__action:
MessageHandler.Msg.ID:='PM115';
MessageHandler.Msg.Name:='Drucker';
MessageHandler.Msg.Text:='Kein Betriebsbereit vom Drucker!Drucker Einschalten weiter mit OK ';
MessageHandler.Msg.Color:=Color.Red;
MessageHandler.Msg.Station:=1;


MessageHandler(
	Prio:=2, 									(*1=highest, .. , 4=lowest*)
	Btn1Addr:=ADR(MsgOk),			(*Address of Button1 , if Zero then Button is unvisible*)
	Btn2Addr:=0,	(*Address of Button2 , if Zero then Button is unvisible*)
	sVisu:=Visu.Message);
END_ACTION

ACTION Msg_Error__exit:
MessageHandler.ClearMessageLines(sVisu:=Visu.Message);
MsgOk:=FALSE;
END_ACTION

ACTION Close_Stopper_action:
ST00_74_Y2_4.MoveInit:=TRUE;
END_ACTION

ACTION WaitForAutoRun_entry:
ST03_Autostop.Start:=FALSE;
END_ACTION

ACTION WaitForAutoRun_action:
IF 	(ModeSelect.Mode=MODE_AUTO_RUN OR
	ModeSelect.Mode=MODE_STEP_RUN OR
	(SpecialMode06.State=State_Run AND
	(gTypeCode=312 OR			(*93pol*)
	gTypeCode=499) ) ) AND			(*102pol*)
	NOT gRunEmpty
THEN
	State:=STATE_RUN;
	SFCTimeStart:=TIME();
ELSE
	State:=STATE_WAIT;
	MsgOK:=FALSE;
	MsgCancel:=FALSE;
	SFCRun:=FALSE;
	ST08_Process.Start:=FALSE;
END_IF

IF 	CTR >= MP.ST03.NoOfTestParts THEN
	CTR:=0;
	gTakeTestParts:=FALSE;
	gTakeTestPartsAuto:=FALSE;
END_IF

IF 	CTR2 >= MP.ST02.NoOfDummys THEN
	CTR2:=0;
	MP.ST02.DummyPruefung_93pol := FALSE;
END_IF
END_ACTION

ACTION WaitForAutoRun_exit:
ST03_Autostop.Start:=TRUE;
END_ACTION

ACTION Wait_for_Part_entry:
ProcessMessage01:='';
Delay.IN:=FALSE;
Delay();
END_ACTION

ACTION Wait_for_Part_action:
ProcessMessage01:='1IM10';(*warte auf Teil in Abholpositon*)
Delay(IN:=ST03_Init_AbholPos.RoboPos31 OR ST03_Init_AbholPos.RoboPos35);
Delay.PT:=T#50ms;
END_ACTION

ACTION Wait_for_Part_exit:
ProcessMessage01:='';
END_ACTION

ACTION Robot01_Pos35___action:
Robot01.PosNo:=POS_WT_POS2;
Robot01.PosOffset:=gRobotOffset;
Robot01.Override:=MP.ST00.Override;
Robot01.SetToolOn:=FALSE;
Robot01.SetToolOff:=TRUE;
Robot01.ExecuteMove:=TRUE;
END_ACTION

ACTION Robot01_Pos35___exit:
IF	Result = RESULT_OK THEN
	gRob01GripState:=PART_OK;
ELSE
	gRob01GripState:=PART_NOK;
END_IF
Result:= RESULT_NON;
END_ACTION

ACTION Robot01_Pos31_5_action:
Robot01.PosNo:=POS_WT_POS1;
Robot01.PosOffset:=gRobotOffset;
Robot01.Override:=MP.ST00.Override;
Robot01.SetToolOn:=FALSE;
Robot01.SetToolOff:=TRUE;
Robot01.ExecuteMove:=TRUE;
END_ACTION

ACTION Robot01_Pos31_5_exit:
IF	Result = RESULT_OK THEN
	gRob01GripState:=PART_OK;
ELSE
	gRob01GripState:=PART_NOK;
END_IF
Result:= RESULT_NON;
END_ACTION

ACTION TestParts_Activ__action:
ST03_51_M1.MotorOn:=TRUE;
END_ACTION

ACTION ST08_Pallett_53_entry:
ProcessMessage01:='';
END_ACTION

ACTION ST08_Pallett_53_action:
ProcessMessage01:='1IM7';(*warte Pallette*)
END_ACTION

ACTION ST08_Pallett_53_exit:
ST08_Process.Start:=FALSE;
ProcessMessage01:='';
END_ACTION

ACTION Robot01_POS_PARK__action:
Robot01.PosNo:=POS_PARK;
Robot01.PosOffset:=gRobotOffset;
Robot01.Override:=MP.ST00.Override;
Robot01.SetToolOn:=FALSE;
Robot01.SetToolOff:=TRUE;
Robot01.ExecuteMove:=TRUE;
END_ACTION

